// TIA Portal V21 program export: 0 tag tables, 0 data types, 38 data blocks, 68 code blocks (in call order from the OBs), 32 instance data blocks

DATA_BLOCK "HmiTags"   // DB16
{ S7_Optimized_Access := 'FALSE' }
// stored: AutoNumber false
   VAR
      MasterReset : Bool;
      SystemRestart : Bool;
      ManualModeFAULT : Bool;
      AlarmAck : Bool;
      Hooter : Bool;
      ResetButton : Bool;
      VesselStatus : Int;
      Weight_int : Int;
      Weight_Temp : Real;
      VesselMaxPressure : Real := 5.0;
      CycleDataLog : Bool;
      CyclePrintData : Bool;
      AlarmPath : String := '/media/simatic/data-storage/Reports/Pdf/Alarm.pdf';
      HelpPath : String := ' /media/simatic/data-storage/OPM/R-OPM.pdf';
      AlarmStarTime : DTL;
      AlarmEndTime : DTL;
      EpoxyMMActual { S7_SetPoint := 'True'} : Real;
      PlcHmiComBreak : Bool;
      AuditStartTime : DTL;
      AuditEndTime : DTL;
      AuditPath : String := '/media/simatic/data-storage/Reports/Pdf/Audit.pdf';
      UserAuditStartTime : DTL;
      UserAuditEndTime : DTL;
      UserAuditPath : String := '/media/simatic/data-storage/Reports/Pdf/UserAudit.pdf';
      LF_time_delay : Int;
      JacketRecoveryCycSelected : Bool;
      JacketRecoveryFault : Bool;
      JacketRecoveryCycEnable : Bool;
      pulse : Array[0..14] of Bool;
      BatchDetailsBlankPopup : Bool;
      BatchDetailsBlankPopupAck : Bool;
      AccessTablePath : String := '/media/simatic/data-storage/Reports/Pdf/AccessTable.pdf';
      LoadCellResult : String;
   END_VAR
BEGIN
END_DATA_BLOCK

DATA_BLOCK "LifeBeatMonitor"   // DB153
{ S7_Optimized_Access := 'FALSE' }
// stored: AutoNumber false
   VAR
      CommunicationBits : Word;
      LifeBit : Bool;
      OnlineOfflineBeat : Bool;
      StartupBit : Bool;
   END_VAR
BEGIN
END_DATA_BLOCK

DATA_BLOCK "ModeDb"   // DB100
{ S7_Optimized_Access := 'FALSE' }
// stored: AutoNumber false
   VAR
      Cycle1 { S7_SetPoint := 'True'} : "ModePara";   // PHT
      Cycle2 { S7_SetPoint := 'True'} : "ModePara";   // BATCH
      Cycle3 { S7_SetPoint := 'True'} : "ModePara";   // SIP
      Cycle4 { S7_SetPoint := 'True'} : "ModePara";   // CIP
      Cycle5 { S7_SetPoint := 'True'} : "ModePara";   // LOAD CELL CALIBRATION
      VesselWeight { S7_SetPoint := 'True'} : Real;
      AlarmStarTime : DTL;
      AlarmEndTime : DTL;
   END_VAR
BEGIN
   Cycle2.CycleName := 'BATCH';
   Cycle3.CycleName := 'SIP';
   Cycle4.CycleName := 'CIP';
   Cycle5.CycleName := 'BULKSTRL';
END_DATA_BLOCK

DATA_BLOCK "ModeDb_R"   // DB110
{ S7_Optimized_Access := 'FALSE' }
// stored: AutoNumber false
   VAR RETAIN
      ManualMode : "ManualModePara";   // MANUAL MODE
      RunningCycle { S7_SetPoint := 'True'} : "CycleDetails";
      BaseReportPath : String := '/media/simatic/data-storage/Reports/Pdf/';
      FinalReportPath : String;
      ReportId : Int;
      Cycle1 { S7_SetPoint := 'True'} : "ModeParaR";   // PHT
      Cycle2 { S7_SetPoint := 'True'} : "ModeParaR";   // BATCH
      Cycle3 { S7_SetPoint := 'True'} : "ModeParaR";   // SIP
      Cycle4 { S7_SetPoint := 'True'} : "ModeParaR";   // CIP
      Cycle5 { S7_SetPoint := 'True'} : "ModeParaR";   // LOAD CELL CALIBRATION
      ReportName : String[100];
   END_VAR
BEGIN
   RunningCycle.PrintInterval := 30;
END_DATA_BLOCK

DATA_BLOCK "ProcessAlarms"   // DB191
{ S7_Optimized_Access := 'FALSE' }
// stored: AutoNumber false
   VAR
      CipCycleOver : Bool;
      CipCycleConductivityReached : Bool;
      CipCycleConductivityNotReached : Bool;
      ConductivityNotSampled : Bool;
      CipReportDataNotLogged : Bool;
      PhtFailed : Bool;
      PhtPassed : Bool;
      PhtOver : Bool;
      PhtReportDataNotLogged : Bool;
      SterilizationTimeOver : Bool;
      SteamFlowLow : Bool;
      SterilizationHighTemperature : Bool;
      SterilizationCycleCompleted : Bool;
      SterilizationReportDataNotLogged : Bool;
      WfiFlowLow : Bool;
      BatchWfiFlowLow : Bool;
   END_VAR
BEGIN
END_DATA_BLOCK

DATA_BLOCK "SafetyAlarms"   // DB181
{ S7_Optimized_Access := 'FALSE' }
// stored: AutoNumber false
   VAR
      ControlKeyOff : Bool;
      EmergencyStopPressed : Bool;
      PowerReset : Bool;
      CompresseDairPressurelow : Bool;
      PowerFailure : Bool;
      PlcRestarted : Bool;
      Mm01FeedbackTrip : Bool;
      Cp01FeedbackTrip : Bool;
      Mm01OverloadTrip : Bool;
      Cp01OverloadTrip : Bool;
      MinimumWeightRequiredToStartmm01 : Bool;
      Ticr01WireBreak : Bool;
      Ticr02WireBreak : Bool;
      Ticr03WireBreak : Bool;
      Ticr04WireBreak : Bool;
      Ticr05WireBreak : Bool;
      Ticr06WireBreak : Bool;
      Ticr07WireBreak : Bool;
      Ticr08WireBreak : Bool;
      Ticr09WireBreak : Bool;
      Ticr10WireBreak : Bool;
      Picr01WireBreak : Bool;
      Picr02WireBreak : Bool;
      Picr03WireBreak : Bool;
      Picr04WireBreak : Bool;
      Cicr01WireBreak : Bool;
      Lc01CommunicationFailed : Bool;
      VesselHighPressure : Bool;
      Mm01SpeedSensorTrip : Bool;
      PlcToHmiCommunicationFailed : Bool;
   END_VAR
BEGIN
END_DATA_BLOCK

DATA_BLOCK "TimerAlarm"   // DB185
{ S7_Optimized_Access := 'FALSE' }
// stored: AutoNumber false
   VAR
      ControlKeyOff : IEC_TIMER;
      EmergencyStopPressed : IEC_TIMER;
      PowerReset : IEC_TIMER;
      CompresseDairPressurelow : IEC_TIMER;
      PowerFailure : IEC_TIMER;
      PlcRestarted : IEC_TIMER;
      Mm01FeedbackTrip : IEC_TIMER;
      Cp01FeedbackTrip : IEC_TIMER;
      Mm01OverloadTrip : IEC_TIMER;
      Cp01OverloadTrip : IEC_TIMER;
      MinimumWeightRequiredToStartmm01 : IEC_TIMER;
      Ticr01WireBreak : IEC_TIMER;
      Ticr02WireBreak : IEC_TIMER;
      Ticr03WireBreak : IEC_TIMER;
      Ticr04WireBreak : IEC_TIMER;
      Ticr05WireBreak : IEC_TIMER;
      Ticr06WireBreak : IEC_TIMER;
      Ticr07WireBreak : IEC_TIMER;
      Ticr08WireBreak : IEC_TIMER;
      Ticr09WireBreak : IEC_TIMER;
      Ticr10WireBreak : IEC_TIMER;
      Picr01WireBreak : IEC_TIMER;
      Picr02WireBreak : IEC_TIMER;
      Picr03WireBreak : IEC_TIMER;
      Picr04WireBreak : IEC_TIMER;
      Cicr01WireBreak : IEC_TIMER;
      Lc01CommunicationFailed : IEC_TIMER;
      VesselHighPressure : IEC_TIMER;
      Mm01SpeedSensorTrip : IEC_TIMER;
      PlcToHmiCommunicationFailed : IEC_TIMER;
      CipCycleOver : IEC_TIMER;
      CipCycleConductivityReached : IEC_TIMER;
      CipCycleConductivityNotReached : IEC_TIMER;
      ConductivityNotSampled : IEC_TIMER;
      CipReportDataNotLogged : IEC_TIMER;
      PhtFailed : IEC_TIMER;
      PhtPass : IEC_TIMER;
      PhtOver : IEC_TIMER;
      PhtReportDataNotLogged : IEC_TIMER;
      SterilizationTimeOver : IEC_TIMER;
      SteamFlowLow : IEC_TIMER;
      SterilizationHighTemperature : IEC_TIMER;
      SterilizationCycleCompleted : IEC_TIMER;
      SterilizationReportDataNotLogged : IEC_TIMER;
      WfiFlowLow : IEC_TIMER;
      BatchReportDataNotLogged : IEC_TIMER;
      LifeBitAlarm { S7_SetPoint := 'True'} : IEC_TIMER;
      AlarmAck_Reset { S7_SetPoint := 'True'} : IEC_TIMER;
      MasterReset { S7_SetPoint := 'True'} : IEC_TIMER;
   END_VAR
BEGIN
END_DATA_BLOCK

DATA_BLOCK "pulse"   // DB8
{ S7_Optimized_Access := 'FALSE' }
   VAR
      ControlKeyOff : Bool;
      EmergencyStopPressed : Bool;
      PowerReset : Bool;
      CompresseDairPressurelow : Bool;
      PowerFailure : Bool;
      PlcRestarted : Bool;
      Mm01FeedbackTrip : Bool;
      Cp01FeedbackTrip : Bool;
      Mm01OverloadTrip : Bool;
      Cp01OverloadTrip : Bool;
      MinimumWeightRequiredToStartmm01 : Bool;
      Ticr01WireBreak : Bool;
      Ticr02WireBreak : Bool;
      Ticr03WireBreak : Bool;
      Ticr04WireBreak : Bool;
      Ticr05WireBreak : Bool;
      Ticr06WireBreak : Bool;
      Ticr07WireBreak : Bool;
      Ticr08WireBreak : Bool;
      Ticr09WireBreak : Bool;
      Ticr10WireBreak : Bool;
      Picr01WireBreak : Bool;
      Picr02WireBreak : Bool;
      Picr03WireBreak : Bool;
      Picr04WireBreak : Bool;
      Cicr01WireBreak : Bool;
      Lc01CommunicationFailed : Bool;
      VesselHighPressure : Bool;
      Mm01SpeedSensorTrip : Bool;
      PlcToHmiCommunicationFailed : Bool;
      CipCycleOver : Bool;
      CipCycleConductivityReached : Bool;
      CipCycleConductivityNotReached : Bool;
      ConductivityNotSampled : Bool;
      CipReportDataNotLogged : Bool;
      PhtFailed : Bool;
      PhtPass : Bool;
      PhtOver : Bool;
      PhtReportDataNotLogged : Bool;
      SterilizationTimeOver : Bool;
      SteamFlowLow : Bool;
      SterilizationHighTemperature : Bool;
      SterilizationCycleCompleted : Bool;
      SterilizationReportDataNotLogged : Bool;
      WfiFlowLow : Bool;
      BatchReportDataNotLogged : Bool;
   END_VAR
BEGIN
END_DATA_BLOCK

DATA_BLOCK "BatchRe"   // DB33
{ S7_Optimized_Access := 'TRUE' }
// stored: AutoNumber false, MemoryReserve 100
   VAR
      ReBit : Array[0..20] of Bool;
      BatchLinePrint : Array[0..60] of String;
   END_VAR
BEGIN
   BatchLinePrint[1] := 'BATCH STARTED';
   BatchLinePrint[2] := 'BATCH OVER';
   BatchLinePrint[3] := 'FILL WFI STARTED';
   BatchLinePrint[4] := 'FILL WFI PAUSED';
   BatchLinePrint[5] := 'FILL WFI RESUMED';
   BatchLinePrint[6] := 'FILL WFI OVER';
   BatchLinePrint[7] := 'FILL WFI RESET';
   BatchLinePrint[8] := 'TEMPERATURE CONTROL HEATING STARTED';
   BatchLinePrint[9] := 'TEMPERATURE CONTROL COOLING STARTED';
   BatchLinePrint[10] := 'TEMPERATURE CONTROL PAUSED';
   BatchLinePrint[11] := 'TEMPERATURE CONTROL RESUMED';
   BatchLinePrint[12] := 'TEMPERATURE CONTROL HEATING REACHED';
   BatchLinePrint[13] := 'TEMPERATURE CONTROL RESET';
   BatchLinePrint[14] := 'MM01 MIXING STARTED';
   BatchLinePrint[15] := 'MM01 MIXING PAUSED';
   BatchLinePrint[16] := 'MM01 MIXING RESUMED';
   BatchLinePrint[17] := 'MM01 MIXING OVER';
   BatchLinePrint[18] := 'MM01 MIXING RESET';
   BatchLinePrint[19] := 'PRODUCT RECIRCULATION STARTED';
   BatchLinePrint[20] := 'PRODUCT RECIRCULATION PAUSED';
   BatchLinePrint[21] := 'PRODUCT RECIRCULATION RESUMED';
   BatchLinePrint[22] := 'PRODUCT RECIRCULATION OVER';
   BatchLinePrint[23] := 'PRODUCT RECIRCULATION RESET';
   BatchLinePrint[24] := 'MANUAL RM ADDITION STARTED';
   BatchLinePrint[25] := 'MANUAL RM ADDITION PAUSED';
   BatchLinePrint[26] := 'MANUAL RM ADDITION RESUMED';
   BatchLinePrint[27] := 'MANUAL RM ADDITION OVER';
   BatchLinePrint[28] := 'MANUAL RM ADDITION RESET';
   BatchLinePrint[29] := 'N2 SPARGING STARTED';
   BatchLinePrint[30] := 'N2 SPARGING PAUSED';
   BatchLinePrint[31] := 'N2 SPARGING RESUMED';
   BatchLinePrint[32] := 'N2 SPARGING OVER';
   BatchLinePrint[33] := 'N2 SPARGING RESET';
   BatchLinePrint[34] := 'GAS BLANKETING STARTED';
   BatchLinePrint[35] := 'GAS BLANKETING PAUSED';
   BatchLinePrint[36] := 'GAS BLANKETING RESUMED';
   BatchLinePrint[37] := 'GAS BLANKETING RESET';
   BatchLinePrint[38] := 'FINAL VOLUME MAKEUP STARTED';
   BatchLinePrint[39] := 'FINAL VOLUME MAKEUP PAUSED';
   BatchLinePrint[40] := 'FINAL VOLUME MAKEUP RESUMED';
   BatchLinePrint[41] := 'FINAL VOLUME MAKEUP OVER';
   BatchLinePrint[42] := 'FINAL VOLUME MAKEUP RESET';
   BatchLinePrint[43] := 'PRODUCT TRANSFER STARTED';
   BatchLinePrint[44] := 'PRODUCT TRANSFER PAUSED';
   BatchLinePrint[45] := 'PRODUCT TRANSFER RESUMED';
   BatchLinePrint[46] := 'PRODUCT TRANSFER OVER';
   BatchLinePrint[47] := 'PRODUCT TRANSFER RESET';
   BatchLinePrint[48] := 'JACKET VENT OPEN';
   BatchLinePrint[49] := 'JACKET VENT CLOSE';
   BatchLinePrint[50] := 'JACKET DRAIN OPEN';
   BatchLinePrint[51] := 'JACKET DRAIN CLOSE';
   BatchLinePrint[52] := 'TEMPERATURE CONTROL COOLING REACHED';
   BatchLinePrint[53] := '-';
END_DATA_BLOCK

DATA_BLOCK "BatchSAD"   // DB301
{ S7_Optimized_Access := 'FALSE' }
// stored: AutoNumber false
   VAR RETAIN
      BatchStart : Bool;
      BatchEnd : Bool;
      BatchStartPopup : Bool;
      BatchStartPopupYes : Bool;
      BatchStartPopupNo : Bool;
      BatchEndPopup : Bool;
      BatchEndPopupYes : Bool;
      BatchEndPopupNo : Bool;
      Fault : Bool;
      RmAddVesselSafetyPressurePopup : Bool;
      BatchEventString : String;
      BatchStartPopup2 : Bool;
      BatchStartPopup2Ack : Bool;
      ProdTransferFilterSel : Int;   // 0 - FILTER BYPASS 1- THROUGH PF01 2- THROUGH PF02
   END_VAR
BEGIN
END_DATA_BLOCK

DATA_BLOCK "BatchTimer"   // DB315
{ S7_Optimized_Access := 'TRUE' }
// stored: AutoNumber false, MemoryReserve 100
   VAR
      Timer01 : IEC_TIMER;
      Timer02 { S7_SetPoint := 'True'} : IEC_TIMER;
      Timer03 { S7_SetPoint := 'True'} : IEC_TIMER;
      Timer04 { S7_SetPoint := 'True'} : IEC_TIMER;
      Timer05 { S7_SetPoint := 'True'} : IEC_TIMER;
      Timer06 { S7_SetPoint := 'True'} : IEC_TIMER;
      Timer07 { S7_SetPoint := 'True'} : IEC_TIMER;
      Timer08 { S7_SetPoint := 'True'} : IEC_TIMER;
      Timer09 { S7_SetPoint := 'True'} : IEC_TIMER;
      Timer10 { S7_SetPoint := 'True'} : IEC_TIMER;
      Timer11 { S7_SetPoint := 'True'} : IEC_TIMER;
      Timer12 { S7_SetPoint := 'True'} : IEC_TIMER;
      Timer13 { S7_SetPoint := 'True'} : IEC_TIMER;
      Timer14 { S7_SetPoint := 'True'} : IEC_TIMER;
      Timer15 { S7_SetPoint := 'True'} : IEC_TIMER;
      Timer16 { S7_SetPoint := 'True'} : IEC_TIMER;
      Timer17 { S7_SetPoint := 'True'} : IEC_TIMER;
      Timer18 { S7_SetPoint := 'True'} : IEC_TIMER;
      Timer19 { S7_SetPoint := 'True'} : IEC_TIMER;
      Timer20 { S7_SetPoint := 'True'} : IEC_TIMER;
      Timer21 { S7_SetPoint := 'True'} : IEC_TIMER;
      Timer22 { S7_SetPoint := 'True'} : IEC_TIMER;
      Timer23 { S7_SetPoint := 'True'} : IEC_TIMER;
      Timer24 { S7_SetPoint := 'True'} : IEC_TIMER;
      Timer25 { S7_SetPoint := 'True'} : IEC_TIMER;
      Timer26 { S7_SetPoint := 'True'} : IEC_TIMER;
      Timer27 { S7_SetPoint := 'True'} : IEC_TIMER;
      Timer28 { S7_SetPoint := 'True'} : IEC_TIMER;
      Timer29 { S7_SetPoint := 'True'} : IEC_TIMER;
      Timer30 { S7_SetPoint := 'True'} : IEC_TIMER;
      Timer31 { S7_SetPoint := 'True'} : IEC_TIMER;
      Timer32 { S7_SetPoint := 'True'} : IEC_TIMER;
      Timer33 { S7_SetPoint := 'True'} : IEC_TIMER;
      Timer34 { S7_SetPoint := 'True'} : IEC_TIMER;
      Timer35 { S7_SetPoint := 'True'} : IEC_TIMER;
      Timer36 { S7_SetPoint := 'True'} : IEC_TIMER;
      Timer37 { S7_SetPoint := 'True'} : IEC_TIMER;
      Timer38 { S7_SetPoint := 'True'} : IEC_TIMER;
      Timer39 { S7_SetPoint := 'True'} : IEC_TIMER;
      Timer40 { S7_SetPoint := 'True'} : IEC_TIMER;
      Timer41 { S7_SetPoint := 'True'} : IEC_TIMER;
      Timer42 { S7_SetPoint := 'True'} : IEC_TIMER;
      Timer43 { S7_SetPoint := 'True'} : IEC_TIMER;
      Timer44 { S7_SetPoint := 'True'} : IEC_TIMER;
      Timer45 { S7_SetPoint := 'True'} : IEC_TIMER;
      Timer46 { S7_SetPoint := 'True'} : IEC_TIMER;
      Timer47 { S7_SetPoint := 'True'} : IEC_TIMER;
      Timer48 { S7_SetPoint := 'True'} : IEC_TIMER;
      Timer49 { S7_SetPoint := 'True'} : IEC_TIMER;
      Timer50 { S7_SetPoint := 'True'} : IEC_TIMER;
      Timer51 { S7_SetPoint := 'True'} : IEC_TIMER;
      Timer52 { S7_SetPoint := 'True'} : IEC_TIMER;
      Timer53 { S7_SetPoint := 'True'} : IEC_TIMER;
      Timer54 { S7_SetPoint := 'True'} : IEC_TIMER;
      Timer55 { S7_SetPoint := 'True'} : IEC_TIMER;
      Timer56 { S7_SetPoint := 'True'} : IEC_TIMER;
      Timer57 { S7_SetPoint := 'True'} : IEC_TIMER;
      Timer58 { S7_SetPoint := 'True'} : IEC_TIMER;
      Timer59 { S7_SetPoint := 'True'} : IEC_TIMER;
      Timer60 { S7_SetPoint := 'True'} : IEC_TIMER;
      Timer61 { S7_SetPoint := 'True'} : IEC_TIMER;
      Timer62 { S7_SetPoint := 'True'} : IEC_TIMER;
      Timer63 { S7_SetPoint := 'True'} : IEC_TIMER;
      Timer64 { S7_SetPoint := 'True'} : IEC_TIMER;
      Timer65 { S7_SetPoint := 'True'} : IEC_TIMER;
   END_VAR
BEGIN
END_DATA_BLOCK

DATA_BLOCK "CipDo"   // DB202
{ S7_Optimized_Access := 'FALSE' }
// stored: AutoNumber false
   VAR
      MM01CmdMagneticMixerMvCommand : Bool;
      CP01CmdCentrifugalPumpMvAreaCommand : Bool;
      HTR01HooterMvArea : Bool;
      LF01VesselLampOutputMv1000 : Bool;
      SPARE4 : Bool;
      SPARE5 : Bool;
      SPARE6 : Bool;
      SPARE7 : Bool;
   END_VAR
BEGIN
END_DATA_BLOCK

DATA_BLOCK "CipPulse"   // DB204
{ S7_Optimized_Access := 'FALSE' }
// stored: AutoNumber false
   VAR
      RE : Array[0..25] of Bool;
      D500EventsTimer : Array[0..25] of IEC_TIMER;
   END_VAR
BEGIN
END_DATA_BLOCK

DATA_BLOCK "CipTimer"   // DB637
{ S7_Optimized_Access := 'TRUE' }
// stored: AutoNumber false, MemoryReserve 100
   VAR
      Timer1 : IEC_TIMER;
      Timer2 { S7_SetPoint := 'True'} : IEC_TIMER;
      Timer3 { S7_SetPoint := 'True'} : IEC_TIMER;
      Timer4 { S7_SetPoint := 'True'} : IEC_TIMER;
      Timer5 { S7_SetPoint := 'True'} : IEC_TIMER;
   END_VAR
BEGIN
END_DATA_BLOCK

DATA_BLOCK "DateTime"   // DB118
{ S7_Optimized_Access := 'FALSE' }
// stored: AutoNumber false
   VAR
      time_local_read : DTL;
      time_system_read : DTL;
      time_system_write : DTL;
      local_time : Int := 0;
      read_system_time : Int;
      write_system_time : Int;
      write_time : Bool := false;
      write_time_re : Bool;
      time_local_read_ReportName : DTL;
   END_VAR
BEGIN
END_DATA_BLOCK

DATA_BLOCK "RTC_to_String_Conversion Block"   // DB119
{ S7_Optimized_Access := 'TRUE' }
// stored: AutoNumber false, MemoryReserve 100
   VAR
      date_int : Int;
      date_string : String[6];
      month_int : Int;
      month_string : String[6];
      year_string : String[6];
      hour_int : Int;
      hour_string : String[6];
      minute_int : Int;
      minute_string : String[6];
      second_int : Int;
      second_string : String[6];
      date_temp : String[6];
      date_zero : Int;
      date_actual : String[12];
      month_temp : String[6];
      month_zero : Int;
      month_actual : String[6];
      year_actual : String[6];
      hour_temp : String[6];
      hour_zero : Int;
      hour_actual : String[6];
      minute_temp : String[6];
      minute_zero : Int;
      minute_actual : String[6];
      second_temp : String[6];
      second_zero : Int;
      second_actual : String[12];
      Final_Date : String[12];
      Final_time_HRS : String[12];
      Final_time_MINS : String[12];
      Final_time_1 : String[12];
      Final_time : String[8];
      SPACE : String[10];
   END_VAR
BEGIN
END_DATA_BLOCK

DATA_BLOCK "Ai_Faceplate_Db"   // DB107
{ S7_Optimized_Access := 'TRUE' }
// stored: AutoNumber false, MemoryReserve 100
   VAR
      Ai01 : "Ai_Faceplate";   // Ticr01NfcoLineTemp
      Ai02 : "Ai_Faceplate";   // Ticr02VfcoLineTemp
      Ai03 : "Ai_Faceplate";   // Ticr03SvcoLineTemp
      Ai04 : "Ai_Faceplate";   // Ticr04VdcoTemp
      Ai05 : "Ai_Faceplate";   // Ticr05CipPumpDrainTemp
      Ai06 : "Ai_Faceplate";   // Ticr06Pf01InLineTemp
      Ai07 : "Ai_Faceplate";   // Ticr07Pf02InLineTemp
      Ai08 : "Ai_Faceplate";   // Ticr08Pf02OutLineTemp
      Ai09 : "Ai_Faceplate";   // Ticr09PtlDrainTemp
      Ai10 : "Ai_Faceplate";   // Ticr10VesselTemp
      Ai11 : "Ai_Faceplate";   // Picr01VesselPressure
      Ai12 : "Ai_Faceplate";   // Picr02VesselRclLine
      Ai13 : "Ai_Faceplate";   // Picr03Pf01OutLinePressure
      Ai14 : "Ai_Faceplate";   // Picr04Pf02OutLinePressure
      Ai15 : "Ai_Faceplate";   // Cicr01ProcessDrainConductivity
      Ai16 : "Ai_Faceplate";   // AiSpare1
      Ai17 : "Ai_Faceplate";   // AiSpare2
      Ai18 : "Ai_Faceplate";   // AiSpare3
      Ai19 : "Ai_Faceplate";   // AiSpare4
      Ai20 : "Ai_Faceplate";   // AiSpare5
      Ai21 : "Ai_Faceplate";   // AiSpare6
      Ai22 : "Ai_Faceplate";   // AiSpare7
      Ai23 : "Ai_Faceplate";   // AiSpare8
      Ai24 : "Ai_Faceplate";   // AiSpare9
      Ai25 : "Ai_Faceplate";
      Ai26 : "Ai_Faceplate";
   END_VAR
BEGIN
END_DATA_BLOCK

DATA_BLOCK "Ao_Faceplate_Db"   // DB105
{ S7_Optimized_Access := 'FALSE' }
// stored: AutoNumber false
   VAR
      Mm01Ref : "Ao_Faceplate";
      Cp01Ref : "Ao_Faceplate";
      Cv01 : "Ao_Faceplate";
      AoSpare1 : "Ao_Faceplate";
      AoSpare2 : "Ao_Faceplate";
      AoSpare3 : "Ao_Faceplate";
      AoSpare4 : "Ao_Faceplate";
      AoSpare5 : "Ao_Faceplate";
   END_VAR
BEGIN
END_DATA_BLOCK

DATA_BLOCK "DO_FaceplateDb"   // DB101
{ S7_Optimized_Access := 'FALSE' }
// stored: AutoNumber false
   VAR
      Cv01 : "Do_Faceplate";
      Cv02 : "Do_Faceplate";
      Cv03 : "Do_Faceplate";
      Cv04 : "Do_Faceplate";
      Cv05 : "Do_Faceplate";
      Cv06 : "Do_Faceplate";
      Cv07 : "Do_Faceplate";
      Cv08 : "Do_Faceplate";
      Cv09 : "Do_Faceplate";
      Cv10 : "Do_Faceplate";
      Cv11 : "Do_Faceplate";
      Cv12 : "Do_Faceplate";
      Cv13 : "Do_Faceplate";
      Cv14 : "Do_Faceplate";
      Cv15 : "Do_Faceplate";
      Cv16 : "Do_Faceplate";
      Cv17 : "Do_Faceplate";
      Cv18 : "Do_Faceplate";
      Cv19 : "Do_Faceplate";
      Cv20 : "Do_Faceplate";
      Cv21 : "Do_Faceplate";
      Cv22 : "Do_Faceplate";
      Cv23 : "Do_Faceplate";
      Cv24 : "Do_Faceplate";
      Cv25 : "Do_Faceplate";
      Cv26 : "Do_Faceplate";
      Cv27 : "Do_Faceplate";
      Cv28 : "Do_Faceplate";
      Cv29 : "Do_Faceplate";
      Cv30 : "Do_Faceplate";
      Cv31 : "Do_Faceplate";
      Cv32 : "Do_Faceplate";
      Cv33 : "Do_Faceplate";
      Cv34 : "Do_Faceplate";
      Cv35 : "Do_Faceplate";
      Cv36 : "Do_Faceplate";
      Cv37 : "Do_Faceplate";
      Cv38 : "Do_Faceplate";
      Cv39 : "Do_Faceplate";
      Cv40 : "Do_Faceplate";
      Cv41 : "Do_Faceplate";
      Cv42 : "Do_Faceplate";
      Cv43 : "Do_Faceplate";
      Cv44 : "Do_Faceplate";
      Cv45 : "Do_Faceplate";
      Cv46 : "Do_Faceplate";
      Cv47 : "Do_Faceplate";
      Cv48 : "Do_Faceplate";
      Cv49 : "Do_Faceplate";
      Cv50 : "Do_Faceplate";
      Cv51 : "Do_Faceplate";
      Cv52 : "Do_Faceplate";
      Cv53 : "Do_Faceplate";
      Cv54 : "Do_Faceplate";
      Cv55 : "Do_Faceplate";
      Cv56 : "Do_Faceplate";
      Cv57 : "Do_Faceplate";
      Cv58 : "Do_Faceplate";
      Cv59 : "Do_Faceplate";
      Cv60 : "Do_Faceplate";
      Cv61 : "Do_Faceplate";
      Cv62 : "Do_Faceplate";
      Cv63 : "Do_Faceplate";
      Cv64 : "Do_Faceplate";
      Fbov01 : "Do_Faceplate";
      "Mm01 Ref" { S7_SetPoint := 'True'} : "Do_Faceplate";
      "Cp01 Ref" { S7_SetPoint := 'True'} : "Do_Faceplate";
   END_VAR
BEGIN
END_DATA_BLOCK

DATA_BLOCK "CV15"   // DB209
{ S7_Optimized_Access := 'TRUE' }
// stored: AutoNumber false, MemoryReserve 100
   VAR
      Tag_IB89 : Byte;
      Tag_IB90 : Byte;
      Tag_IB93 : Byte;
      Tag_IB94 : Byte;
      Tag_IB96 : Byte;
      Tag_IB97 : Byte;
      Tag_IB98 : Byte;
      Tag_MD124 : DInt;
      Tag_MD300 : DInt;
      Tag_MD304 : DInt;
      Tag_MD308 : DInt;
      Tag_MD312 : Real;
      Tag_MD316 : Real;
      Tag_MD320 : DInt;
      Tag_MD324 : DInt;
      Tag_MD340 : DInt;
      Tag_MD344 : DInt;
      Tag_MD348 { ExternalWritable := 'False'} : DInt;
      Tag_MD352 : Real;
      Tag_MD356 : Real;
   END_VAR
BEGIN
END_DATA_BLOCK

DATA_BLOCK "PHT Cycle"   // DB1201
{ S7_Optimized_Access := 'FALSE' }
// stored: AutoNumber false
   VAR
      Start : Bool;
      Stop : Bool;
      Abort : Bool;
      fault : Bool;
      Running : Bool;
      Selected : Bool;
      Actual_Min_Pressure : Real;
      Actual_Max_Pressure : Real;
      "Actual Stabilization Time" : DInt;
      "Actual Pressurise Hold Mins" : DInt;
      "Actual Pressurise Hold Secs" : DInt;
      "PHT Step Status int" : Int;
      "Step Status" : String[50];
      "Event Status" : String[50];
      print_event : Bool;
      "Startup Popup" : Bool;
      "Startup Popup Ack" : Bool;
      "Startup Popup Acked" : Bool;
      "Startup parameter popup" : Bool;
      "Abort Confirmation Popup" : Bool;
      "PHT Result" : Int;
      VesselSel : Int := 1;   // 1=Mv1, 2=Mv2, 3=Mv1&Mv2
      Result : String[50];
      Continue_Button : Bool;
      Abort_Button : Bool;
      "Actual Delay to Open Cai" : Int;
      PhtTemp : Bool;
      HOLD_FAIL : Bool;
      "Startup parameter popup No" : Bool;
      "Startup parameter popup Yes" : Bool;
      "Actual Delay to Open N2I" : Int;
      "N2IControl Valve" : Bool;
      EndOverPopup : Bool;
      EndOverPopupAck : Bool;
      CycleAbortEvent : Bool;
      "Abort confirmation popup Yes" : Bool;
      "Abort confirmation popup No" : Bool;
      InitialPressure : Real;
      FinalPressure : Real;
      HoldStartTimeLog : DTL;
      HoldEndTimeLog : DTL;
      TempTime : Time;
      RoundedTime : Time;
      TempMs : DInt;
      RoundedTime_Pos : Time;
      Hours : Int;
      Minutes : Int;
      Seconds : Int;
      TotalSecondsTag : DInt;
      PhtTimeDifference : Time;
   END_VAR
BEGIN
END_DATA_BLOCK

DATA_BLOCK "PHTRe"   // DB41
{ S7_Optimized_Access := 'TRUE' }
// stored: AutoNumber false, MemoryReserve 100
   VAR
      PhtLinePrintText : Array[0..10] of String[40];
      PhtLinePrint1 : String[40];
      RE : Array[0..20] of Bool;
   END_VAR
BEGIN
   PhtLinePrintText[1] := 'PRESSURIZE STARTED';
   PhtLinePrintText[2] := 'STABILIZE STARTED';
   PhtLinePrintText[3] := 'PRESSURE HOLD STARTED';
   PhtLinePrintText[4] := 'PRESSURE RELEASE STARTED';
   PhtLinePrintText[5] := 'CYCLE PAUSED';
   PhtLinePrintText[6] := 'PHT OVER';
END_DATA_BLOCK

DATA_BLOCK "PhtRecipe"   // DB1218
{ S7_Optimized_Access := 'FALSE' }
// stored: AutoNumber false
   VAR
      HoldPressure : Real := 1.33;
      PressureStabilizeTime : Int := 30;
      AcceptableLeakage : Real := 0.2;
      PressureHoldTime : Int := 1;
      ReleasePressure : Real := 0.1;
   END_VAR
BEGIN
END_DATA_BLOCK

DATA_BLOCK "PhtTimer"   // DB1216
{ S7_Optimized_Access := 'FALSE' }
// stored: AutoNumber false
   VAR
      "ReportData ResetTImer" : IEC_TIMER;
      "TIMER" { S7_SetPoint := 'True'} : IEC_TIMER;
      HVEventsTimer : Array[0..20] of IEC_TIMER;
      PhtTime1 { S7_SetPoint := 'True'} : IEC_TIMER;
      PhtTime2 { S7_SetPoint := 'True'} : IEC_TIMER;
      PhtTime3 { S7_SetPoint := 'True'} : IEC_TIMER;
      PhtTime4 { S7_SetPoint := 'True'} : IEC_TIMER;
      PhtTime5 { S7_SetPoint := 'True'} : IEC_TIMER;
      PhtTime6 { S7_SetPoint := 'True'} : IEC_TIMER;
      PhtTime7 { S7_SetPoint := 'True'} : IEC_TIMER;
      PhtTime8 { S7_SetPoint := 'True'} : IEC_TIMER;
      PhtTime9 { S7_SetPoint := 'True'} : IEC_TIMER;
      PhtTime10 { S7_SetPoint := 'True'} : IEC_TIMER;
   END_VAR
BEGIN
END_DATA_BLOCK

DATA_BLOCK "PidParameters"   // DB58
{ S7_Optimized_Access := 'FALSE' }
   VAR RETAIN
      Fv1_Cv01 : Struct
         "Set Value" : Real;
         P : Real := 8.0;
         I : Real := 80.0;
         D : Real := 0.0;
         Mode : Int;
         Output : Real;
         OutputCoil : Bool;
         State : Int;
         Error : Word;
         Reset : Bool;
         InputValue : Real;
      END_STRUCT;
   END_VAR
BEGIN
END_DATA_BLOCK

DATA_BLOCK "CipRe"   // DB42
{ S7_Optimized_Access := 'TRUE' }
// stored: MemoryReserve 100
   VAR
      CipLinePrintText : Array[0..20] of String;
   END_VAR
BEGIN
   CipLinePrintText[1] := 'PRE RINSE CYCLE - RINSING ON STARTED';
   CipLinePrintText[2] := 'PRE RINSE CYCLE - DRAIN ON STARTED';
   CipLinePrintText[3] := 'PRE RINSE CYCLE - SYSTEM DRAIN STARTED';
   CipLinePrintText[4] := 'PRE RINSE CYCLE - AIR PURGING STARTED';
   CipLinePrintText[5] := 'FILLING CYCLE - FILLING ON STARTED';
   CipLinePrintText[6] := 'FILLING CYCLE - MIXING ON STARTED';
   CipLinePrintText[7] := 'FILLING CYCLE - DRAIN ON STARTED';
   CipLinePrintText[8] := 'FILLING CYCLE - SYSTEM DRAIN STARTED';
   CipLinePrintText[9] := 'FILLING CYCLE - AIR PURGING ON STARTED';
   CipLinePrintText[10] := 'WAITING FOR ACKNOWLEDGE';
   CipLinePrintText[11] := 'CYCLE PAUSED';
   CipLinePrintText[12] := 'CIP CYCLE OVER';
   CipLinePrintText[13] := 'CYCLE RESETED';
   CipLinePrintText[14] := 'FILLING CYCLE - RECIRCULATION STARTED';
   CipLinePrintText[15] := 'FINAL RINSE CYCLE - FILLING ON STARTED';
   CipLinePrintText[16] := 'FINAL RINSE CYCLE - MIXING ON STARTED';
   CipLinePrintText[17] := 'FINAL RINSE CYCLE - DRAIN ON STARTED';
   CipLinePrintText[18] := 'FINAL RINSE CYCLE - SYSTEM DRAIN STARTED';
   CipLinePrintText[19] := 'FINAL RINSE CYCLE - AIR PURGING ON STARTED';
   CipLinePrintText[20] := 'FINAL RINSE CYCLE - RECIRCULATION STARTED';
END_DATA_BLOCK

DATA_BLOCK "DB615"   // DB615
TITLE = DB615
{ S7_Optimized_Access := 'FALSE' }
// CIP GENERAL DB
// stored: AutoNumber false
   VAR RETAIN
      Fault : Bool;
      Running : Bool;
      Selected : Bool;
      NoCycleSelectedInterlock : Bool;
      SelectStep : Bool;
      DelayToTriggerStep : Bool;
      ResetLogic : Bool;
      ProcessOver : Bool;
      TempStep : Int;
      CurrentStep : Int;
      CycleStatus : String[60];
      StepStatus : String[60];
      StepStatusInt : Int;
      Re : Array[0..50] of Bool;
      CycleStarted { S7_SetPoint := 'True'} : "CipCycleStarted";
      CycleOver { S7_SetPoint := 'True'} : "CipCycleOver";
      CycleRunningMV : Bool;
      ApActPressure : Real;
      CheckWeightWfi : Real;
      ScanTimeForFillingWfiTemp : Int;
   END_VAR
BEGIN
END_DATA_BLOCK

DATA_BLOCK "DB621"   // DB621
TITLE = DB619
{ S7_Optimized_Access := 'TRUE' }
// CIP BUTTONS DB
// stored: AutoNumber false, MemoryReserve 0
   VAR
      Start : Bool;
   END_VAR
   VAR RETAIN
      MainPopup1Ack : Bool;
      MainPopup2Ack : Bool;
   END_VAR
BEGIN
END_DATA_BLOCK

DATA_BLOCK "DB622"   // DB622
TITLE = DB620
{ S7_Optimized_Access := 'FALSE' }
// CIP POPUPS
// stored: AutoNumber false
   VAR RETAIN
      NoCycleSelectedPopup : Bool;
      MainPopupMsg1 : Bool;
      MainPopupMsg2 : Bool;
   END_VAR
BEGIN
END_DATA_BLOCK

DATA_BLOCK "DB625"   // DB625
TITLE = REPORT PROCESS VALUE
{ S7_Optimized_Access := 'FALSE' }
// stored: AutoNumber false
   VAR RETAIN
      RepetitionPrint : Array[0..3] of Int;
      FillingPrint : Array[0..3] of "FillingPrint";
      MixingTime { S7_SetPoint := 'True'} : Array[0..3] of "MixingPrint";
      Pulsingtime { S7_SetPoint := 'True'} : Array[0..3] of "PulsingPrint";
      spare { S7_SetPoint := 'True'} : Bool;
      RecirculationPrint { S7_SetPoint := 'True'} : Array[0..3] of "RecirculationPrint";
      DrainPrint { S7_SetPoint := 'True'} : Array[0..3] of "DrainPrint";
      ConductivityStatus { S7_SetPoint := 'True'} : Array[0..3] of Bool;
   END_VAR
BEGIN
END_DATA_BLOCK

DATA_BLOCK "DB626"   // DB626
TITLE = ZERO REPORT PROCESS VALUE
{ S7_Optimized_Access := 'FALSE' }
// stored: AutoNumber false
   VAR
      RepetitionPrint : Array[0..3] of Int;
      FillingPrint : Array[0..3] of "FillingPrint";
      MixingTime { S7_SetPoint := 'True'} : Array[0..3] of "MixingPrint";
      Pulsingtime { S7_SetPoint := 'True'} : Array[0..3] of "PulsingPrint";
      spare { S7_SetPoint := 'True'} : Bool;
      RecirculationPrint { S7_SetPoint := 'True'} : Array[0..3] of "RecirculationPrint";
      DrainPrint { S7_SetPoint := 'True'} : Array[0..3] of "DrainPrint";
      ConductivityStatus { S7_SetPoint := 'True'} : Array[0..3] of Bool;
   END_VAR
BEGIN
END_DATA_BLOCK

DATA_BLOCK "DB627"   // DB627
TITLE = SCREEN PROCESS VALUE
{ S7_Optimized_Access := 'FALSE' }
// stored: AutoNumber false
   VAR
      RinseTimeSv : Int;
      RinseTimePv : DInt;
      FillTimeSv : DInt;
      FillTimePv : DInt;
      RepSv : Int;
      RepPv : Int;
      FillQtySv : Real;
      FillQtyPv : Real;
      MixingSv : Int;
      MixingPv : DInt;
      SdSv : Int;
      SdPv : DInt;
      APSv : Int;
      ApPv : DInt;
      ApReleaseTimeSv : Int;
      ApReleaseTimePv : DInt;
      CurrentStepNo : Int;
      CycleStatus : String[60];
      StepStatus : String[60];
      ApSetPressureSv : Real;
      ApSetPressurePv : Real;
      CombineAPSv : Int;
      CombineApPv : DInt;
      CombineApReleaseTimeSv : Int;
      CombineApReleaseTimePv : DInt;
      DosingTimePv : DInt;
      PulsingTimeSv : Int;
      RecirculationSv : Int;
      RecirculationPv : DInt;
      ConductivitySv : Real;
      ConductivityPv : Real;
   END_VAR
BEGIN
END_DATA_BLOCK

DATA_BLOCK "DB616"   // DB616
TITLE = DB616
{ S7_Optimized_Access := 'FALSE' }
// CIP Recipe
// stored: AutoNumber false
   VAR
      TotalStep : Int := 3;
      CycleSelection { S7_SetPoint := 'True'} : Array[0..3] of "CIP";
      MainPopup1Enable : Bool := 1;
      MainPopup2Enable : Bool := 1;
      FillingInputPara { S7_SetPoint := 'True'} : Array[0..3] of "FillingInputs";
      FillingOutputPara { S7_SetPoint := 'True'} : Array[0..3] of "FillingOutputs";
      MixingTimeInput : Array[0..3] of Int;
      RecirculationInput { S7_SetPoint := 'True'} : Array[0..3] of "RecirculationInputs";
      RecirculationOutput { S7_SetPoint := 'True'} : Array[0..3] of "RecirculationOutputs";
      DrainInputs { S7_SetPoint := 'True'} : Array[0..3] of "DrainInputs";
      DrainOutputs : Array[0..3] of "DrainOutputs";
      SystemDrainSetTimeInput : Array[0..3] of Int;
      SystemDrainOutPara { S7_SetPoint := 'True'} : Array[0..3] of "SystemDrainOutputs";
      AirPurgingInputPara { S7_SetPoint := 'True'} : Array[0..3] of "AirPurgingInputs";
      AirPurgingOutPara { S7_SetPoint := 'True'} : Array[0..3] of "AirPurgingOutputs";
      CycleNames : Array[0..3] of String[60];
      Spare : Bool;
   END_VAR
BEGIN
   CycleSelection[0..3].StepSelection.SuctionLineCleanNoYes := 0;
   CycleSelection[0..3].StepSelection.VacuumDryingNoYes := 0;
   CycleSelection[0].StepSelection.FillingNoYes := 0;
   CycleSelection[1..3].StepSelection.FillingNoYes := 1;
   CycleSelection[0..3].StepSelection.TemperatureDosingNoYes := 0;
   CycleSelection[0..3].StepSelection.TransferNoYes := 0;
   CycleSelection[0..1].StepSelection.MIxingNoYes := 0;
   CycleSelection[2..3].StepSelection.MIxingNoYes := 1;
   CycleSelection[0..1].StepSelection.RecirculationNoYes := 0;
   CycleSelection[2..3].StepSelection.RecirculationNoYes := 1;
   CycleSelection[0].StepSelection.DrainNoYes := 0;
   CycleSelection[1..3].StepSelection.DrainNoYes := 1;
   CycleSelection[0].StepSelection.SystemDrainNoYes := 0;
   CycleSelection[1..3].StepSelection.SystemDrainNoYes := 1;
   CycleSelection[0].StepSelection.AirPurgingNoYes := 0;
   CycleSelection[1..3].StepSelection.AirPurgingNoYes := 1;
   CycleSelection[1..3].StepSelection.ConductivityCheckWhileRinse := 0;
   CycleSelection[0..2].StepSelection.ConductivityCheckWhileDrain := 0;
   CycleSelection[3].StepSelection.ConductivityCheckWhileDrain := 1;
   CycleSelection[0..2].StepSelection.SetRepetition := 0;
   CycleSelection[0..3].StepSelection.TimeSaveModeNoYes := 0;
   CycleSelection[1].StepSelection.ConductivityCheckWhileTransfer := false;
   CycleSelection[2..3].StepSelection.ConductivityCheckWhileTransfer := 0;
   FillingInputPara[1].Selections.FillMethodSel := 3;
   FillingInputPara[2..3].Selections.FillMethodSel := 0;
   FillingInputPara[1..3].Selections.FillTimeBaseSel := 0;
   FillingInputPara[0].Selections.UtilitySel := 1;
   FillingInputPara[1..3].Selections.UtilitySel := 2;
   FillingInputPara[1..3].Selections.ConductivityWhileRinse := 0;
   FillingInputPara[0].Selections.RinseCondition := 1;
   FillingInputPara[1..3].Selections.RinseCondition := 0;
   FillingInputPara[1].Selections.BypassRinseCondition := 1;
   FillingInputPara[2..3].Selections.BypassRinseCondition := 0;
   FillingInputPara[1..3].Selections.BypassWeightWhileRinseCycle := 0;
   FillingInputPara[0..3].Selections.SeperateParaForRep := 1;
   FillingInputPara[1..2].ProductionSetting.LoopDelay1 := 0;
   FillingInputPara[1].ProductionSetting.ZDVDelay := 0;
   FillingInputPara[0].PreciseEngineering.Loops := 1;
   FillingInputPara[1].PreciseEngineering.Loops := 16;
   FillingInputPara[2..3].PreciseEngineering.Loops := 5;
   FillingInputPara[1..3].PreciseEngineering.VesselMaxWeight := 3000.0;
   MixingTimeInput[2..3] := 1;
   RecirculationInput[2..3].Selections.PressureModeSel := 0;
   RecirculationInput[2..3].Selections.PumpSel := 0;
   RecirculationInput[2].Parameters.RecirculationInputToRunTime := 0;
   RecirculationInput[1].PreciseEngineering.Loops := 0;
   RecirculationInput[2..3].PreciseEngineering.Loops := 5;
   DrainInputs[0..3].Selections.DrainMethodSel := 0;
   DrainInputs[1..3].Selections.PressureModeSel := 1;
   DrainInputs[1].Selections.DrainPumpSel := 0;
   DrainInputs[2..3].Selections.DrainPumpSel := 1;
   DrainInputs[0..1].Selections.InputToRunPump := 0;
   DrainInputs[2..3].Selections.InputToRunPump := 1;
   DrainInputs[1..2].Selections.ConductivityWhileDrain := 0;
   DrainInputs[3].Selections.ConductivityWhileDrain := 1;
   DrainInputs[1..2].Selections.ConductivityWhileDrainPTL := 0;
   DrainInputs[1..2].Selections.CipSkidWeightSel := 0;
   DrainInputs[1..2].Selections.MultiConductivityCheck := 0;
   DrainInputs[0..1].PreciseEngineering.Loops := 1;
   DrainInputs[2..3].PreciseEngineering.Loops := 10;
   AirPurgingInputPara[1..3].Selections.ApMethod := 0;
   AirPurgingInputPara[1..3].Selections.PressureMode := 1;
   AirPurgingInputPara[1..3].Selections.VentBeforeOver := 1;
   AirPurgingInputPara[1..3].Selections.AirPurgingSel := 0;
   AirPurgingInputPara[1..3].PreciseEngineering.Loops := 17;
   CycleNames[1] := 'PRE RINSE CYCLE';
   CycleNames[2] := 'FILLING CYCLE';
   CycleNames[3] := 'FINAL RINSE CYCLE';
END_DATA_BLOCK

DATA_BLOCK "DB623"   // DB623
TITLE = DB618
{ S7_Optimized_Access := 'FALSE' }
// Recipe
// stored: AutoNumber false
   VAR RETAIN
      StepEnable : Array[0..5] of Bool;
      Mm01Speed : Real := 1200.0;
      Cp01Speed : Real := 1000.0;
      DrainPressure : Real := 1.11;
      AirPurgingPressure : Real := 1.33;
      SystemDrainTime : Int := 30;
      PreRinseCycleSelection : Int := 1;
      FillingCycleSelection : Int := 1;
      FinalRinseCycleSelection : Int := 1;
      PreRinseCycleNoOfRep : Int := 1;
      FillingCycleNoOfRep : Int := 2;
      FillingCycleMixingTime : Int := 30;
      FinalRinseCycleMixingTime : Int := 35;
      FillingCycleFillQty : Real := 500.0;
      FinalRinseCycleFillQty : Real := 1000.0;
      PreRinseCycleSelString : String[10];
      FillingCycleSelString : String[10];
      FinalRinseCycleSelString : String[10];
      FinalRinseSetCond : Real := 1.22;
      SbiOnTime : Int := 10;
      SbiOffTime : Int := 5;
   END_VAR
BEGIN
   StepEnable[0] := FALSE;
   StepEnable[1..3] := TRUE;
END_DATA_BLOCK

DATA_BLOCK "DB624"   // DB624
{ S7_Optimized_Access := 'FALSE' }
// stored: AutoNumber false
   VAR RETAIN
      PcdTime : Int := 10;
      VesselDrainWeight : Real := 15.0;
      AirPurgingPressureTolerence : Real := 0.1;
      AirPurgingReleaseTime : Int := 30;
      DrainPressureTolerance : Real := 0.2;
      DelayToCheckConductivity : Int := 10;
      ConductivityCheckTime : Int := 5;
      "FinalRinseCycleNo.OfRep" : Int := 3;
      FillRinseSamplingLineDelay : Int := 30;
      FillRinseBlanketingLineDelay : Int := 30;
      FillRinseJTubeLineDelay : Int := 30;
      FillRinseSpargingLineDelay : Int := 30;
      FillRinseSbiLineDelay : Int := 30;
      FillRinseRecirculationlineDelay : Int := 30;
      FillRinseVesselBypassLineDelay : Int := 30;
      FillRinsePumpBypassLineDelay : Int := 30;
      FillRinsePf01InLineDelay : Int := 30;
      FillRinsePf01VentLineDelay : Int := 30;
      FillRinsePf02InLineDelay : Int := 30;
      FillRinsePf02VentLineDelay : Int := 30;
      FillRinsePf02OutLineDelay : Int := 30;
      FillRinsePf01BypassLineDelay : Int := 30;
      FillRinsePf02BypassLineDelay : Int := 30;
      FillRinsePtlLineDelay : Int := 30;
      RecSamplingLineDelay : Int := 30;
      RecBlanketingLineDelay : Int := 30;
      RecJTubeLineDelay : Int := 30;
      RecSpargingLineDelay : Int := 30;
      RecSbiLineDelay : Int := 30;
      DrainVesselDrainLineDelay : Int := 30;
      DrainPumpBypassLineDelay : Int := 30;
      DrainPf01InLineDelay : Int := 30;
      DrainPf01VentLineDelay : Int := 30;
      DrainPf02InLineDelay : Int := 30;
      DrainPf02VentLineDelay : Int := 30;
      DrainPf02OutLineDelay : Int := 30;
      DrainPf01BypassLineDelay : Int := 30;
      DrainPf02BypassLineDelay : Int := 30;
      FinalRinseCycleVesselDrainLineDelay : Int := 30;
      AirPurgeSamplingLineDelay : Int := 30;
      AirPurgeBlankeingLineDelay : Int := 30;
      AirPurgeJTubeLineDelay : Int := 30;
      AirPurgeSpargingLineDelay : Int := 30;
      AirPurgeSbiLineDelay : Int := 30;
      AirPurgeRecirculationlineDelay : Int := 30;
      AirPurgeVesselBypassLineDelay : Int := 30;
      AirPurgeVesselDrainLineDelay : Int := 30;
      AirPurgePumpBypassLineDelay : Int := 30;
      AirPurgePf01InLineDelay : Int := 30;
      AirPurgePf01VentLineDelay : Int := 30;
      AirPurgePf02InLineDelay : Int := 30;
      AirPurgePf02VentLineDelay : Int := 30;
      AirPurgePf02OutLineDelay : Int := 30;
      AirPurgePf01BypassLineDelay : Int := 30;
      AirPurgePf02BypassLineDelay : Int := 30;
      AirPurgePtlLineDelay : Int := 30;
   END_VAR
BEGIN
END_DATA_BLOCK

DATA_BLOCK "DiFinal"   // DB102
{ S7_Optimized_Access := 'FALSE' }
// stored: AutoNumber false
   VAR
      ControlKey : Bool;
      EmergencyStop : Bool;
      CompressedAirPressureLow : Bool;
      PowerFailure : Bool;
      PowerReset : Bool;
      MagneticMixerFeedback : Bool;
      CipPumpFeedback : Bool;
      MagneticMixerOverload : Bool;
      CipPumpOverload : Bool;
      RuptureDisc : Bool;
      Cp01FlowSwitch : Bool;
      DiSpare1 : Bool;
      DiSpare2 : Bool;
      MMHighSpeedSensor : Bool;
      DiSpare3 : Bool;
      DiSpare4 : Bool;
      DiSpare5 : Bool;
      DiSpare6 : Bool;
      DiSpare7 : Bool;
      DiSpare8 : Bool;
      DiSpare9 : Bool;
      DiSpare10 : Bool;
   END_VAR
BEGIN
END_DATA_BLOCK

DATA_BLOCK "DiSimulation"   // DB103
{ S7_Optimized_Access := 'TRUE' }
// stored: AutoNumber false, MemoryReserve 100
   VAR
      ControlKey : Bool;
      EmergencyStop : Bool;
      CompressedAirPressureLow : Bool;
      PowerFailure : Bool;
      PowerReset : Bool;
      MagneticMixerFeedback : Bool;
      CipPumpFeedback : Bool;
      MagneticMixerOverload : Bool;
      CipPumpOverload : Bool;
      RuptureDisc : Bool;
      Cp01FlowSwitch : Bool;
      DiSpare1 : Bool;
      DiSpare2 : Bool;
      MMHighSpeedSensor : Bool;
      DiSpare3 : Bool;
      DiSpare4 : Bool;
      DiSpare5 : Bool;
      DiSpare6 : Bool;
      DiSpare7 : Bool;
      DiSpare8 : Bool;
      DiSpare9 : Bool;
      DiSpare10 : Bool;
   END_VAR
BEGIN
END_DATA_BLOCK

DATA_BLOCK "DoManualModeDb"   // DB2
{ S7_Optimized_Access := 'FALSE' }
// stored: AutoNumber false
   VAR
      Mm01Cmd : Bool;
      Cp01Cmd : Bool;
      Htr : Bool;
      Lf01 : Bool;
      DoSpare1 : Bool;
      DoSpare2 : Bool;
      DoSpare3 : Bool;
      DoSpare4 : Bool;
      DoSpare5 : Bool;
      DoSpare6 : Bool;
   END_VAR
BEGIN
END_DATA_BLOCK

ORGANIZATION_BLOCK "Main"   // OB1, LAD, ProgramCycle
TITLE = "Main Program Sweep (Cycle)"
{ S7_Optimized_Access := 'TRUE' }
// stored: SetENOAutomatically false
   VAR_INPUT
      Initial_Call : Bool;   // Initial call of this OB
      Remanence : Bool;   // =True, if remanent data are available
   END_VAR
   VAR_TEMP   // added for the SCL form of the ladder/FBD networks
      _w1 : Bool;
   END_VAR
BEGIN

REGION Network 1: "Sec_Pulse"
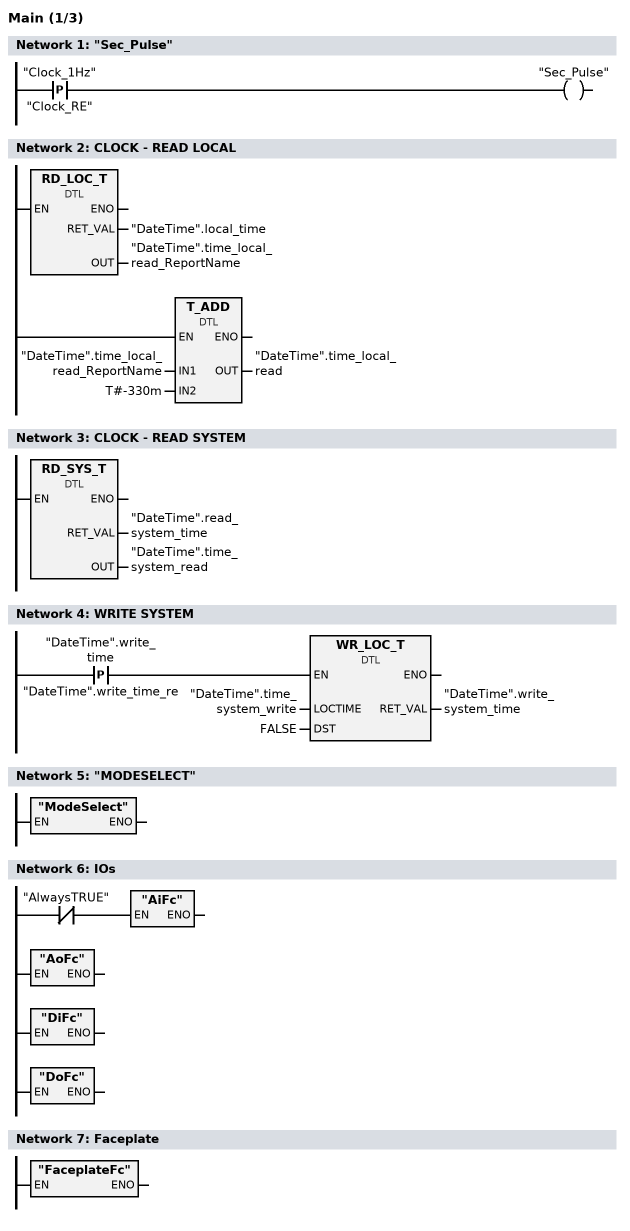
   RUNG wire#powerrail
      P_Contact(operand := "Clock_1Hz", bit := "Clock_RE")
      Coil( "Sec_Pulse" )
   END_RUNG
   // the same network as SCL:
   #_w1 := "Clock_1Hz" AND NOT "Clock_RE";   // rising edge of "Clock_1Hz"
   "Clock_RE" := "Clock_1Hz";
   "Sec_Pulse" := #_w1;
END_REGION

REGION Network 2: CLOCK - READ LOCAL
   RUNG wire#powerrail
      { S7_Templates := "date_type := DTL" } RD_LOC_T(RET_VAL => "DateTime".local_time, OUT => "DateTime".time_local_read_ReportName)
   END_RUNG
   RUNG wire#powerrail
      { S7_Templates := "[date_type := DTL, time_type := Time]" } T_ADD(IN1 := "DateTime".time_local_read_ReportName, IN2 := T#-330m, OUT => "DateTime".time_local_read)
   END_RUNG
   // the same network as SCL:
   "DateTime".local_time := RD_LOC_T(OUT => "DateTime".time_local_read_ReportName);
   T_ADD(IN1 := "DateTime".time_local_read_ReportName, IN2 := T#-330m, OUT => "DateTime".time_local_read);
END_REGION

REGION Network 3: CLOCK - READ SYSTEM
   RUNG wire#powerrail
      { S7_Templates := "date_type := DTL" } RD_SYS_T(RET_VAL => "DateTime".read_system_time, OUT => "DateTime".time_system_read)
   END_RUNG
   // the same network as SCL:
   "DateTime".read_system_time := RD_SYS_T(OUT => "DateTime".time_system_read);
END_REGION

REGION Network 4: WRITE SYSTEM
   RUNG wire#powerrail
      P_Contact(operand := "DateTime".write_time, bit := "DateTime".write_time_re)
      { S7_Templates := "loctime_type := DTL" } WR_LOC_T(LOCTIME := "DateTime".time_system_write, DST := FALSE, Ret_Val => "DateTime".write_system_time)
   END_RUNG
   // the same network as SCL:
   #_w1 := "DateTime".write_time AND NOT "DateTime".write_time_re;   // rising edge of "DateTime".write_time
   "DateTime".write_time_re := "DateTime".write_time;
   IF #_w1 THEN
       "DateTime".write_system_time := WR_LOC_T(LOCTIME := "DateTime".time_system_write, DST := FALSE);
   END_IF;
END_REGION

REGION Network 5: "MODESELECT"
   RUNG wire#powerrail
      "ModeSelect"()
   END_RUNG
   // the same network as SCL:
   "ModeSelect"();
END_REGION

REGION Network 6: IOs
   RUNG wire#powerrail
      I_Contact( "AlwaysTRUE" )
      "AiFc"()
   END_RUNG
   RUNG wire#powerrail
      "AoFc"()
   END_RUNG
   RUNG wire#powerrail
      "DiFc"()
   END_RUNG
   RUNG wire#powerrail
      "DoFc"()
   END_RUNG
   // the same network as SCL:
   IF NOT "AlwaysTRUE" THEN "AiFc"(); END_IF;
   "AoFc"();
   "DiFc"();
   "DoFc"();
END_REGION

REGION Network 7: Faceplate
   RUNG wire#powerrail
      "FaceplateFc"()
   END_RUNG
   // the same network as SCL:
   "FaceplateFc"();
END_REGION

REGION Network 8: ValvesOutputFc
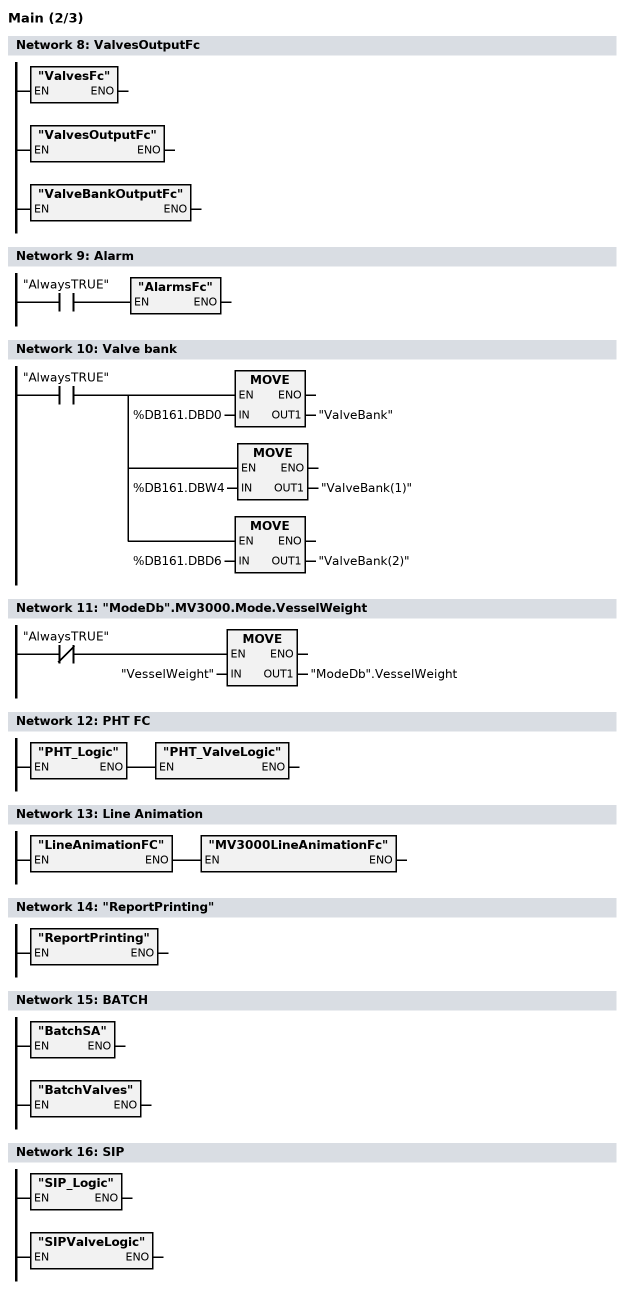
   RUNG wire#powerrail
      "ValvesFc"()
   END_RUNG
   RUNG wire#powerrail
      "ValvesOutputFc"()
   END_RUNG
   RUNG wire#powerrail
      "ValveBankOutputFc"()
   END_RUNG
   // the same network as SCL:
   "ValvesFc"();
   "ValvesOutputFc"();
   "ValveBankOutputFc"();
END_REGION

REGION Network 9: Alarm
   RUNG wire#powerrail
      Contact( "AlwaysTRUE" )
      "AlarmsFc"()
   END_RUNG
   // the same network as SCL:
   IF "AlwaysTRUE" THEN "AlarmsFc"(); END_IF;
END_REGION

REGION Network 10: Valve bank
   RUNG wire#powerrail
      Contact( "AlwaysTRUE" )
      wire#w1
      Move(in := %DB161.DBD0, out1 => "ValveBank")
   END_RUNG
   RUNG wire#w1
      Move(in := %DB161.DBW4, out1 => "ValveBank(1)")
   END_RUNG
   RUNG wire#w1
      Move(in := %DB161.DBD6, out1 => "ValveBank(2)")
   END_RUNG
   // the same network as SCL:
   IF "AlwaysTRUE" THEN
       "ValveBank" := %DB161.DBD0;
       "ValveBank(1)" := %DB161.DBW4;
       "ValveBank(2)" := %DB161.DBD6;
   END_IF;
END_REGION

REGION Network 11: "ModeDb".MV3000.Mode.VesselWeight
   RUNG wire#powerrail
      I_Contact( "AlwaysTRUE" )
      Move(in := "VesselWeight", out1 => "ModeDb".VesselWeight)
   END_RUNG
   // the same network as SCL:
   IF NOT "AlwaysTRUE" THEN "ModeDb".VesselWeight := "VesselWeight"; END_IF;
END_REGION

REGION Network 12: PHT FC
   RUNG wire#powerrail
      "PHT_Logic"()
      "PHT_ValveLogic"()
   END_RUNG
   // the same network as SCL:
   "PHT_Logic"(ENO => #_w1);
   IF #_w1 THEN "PHT_ValveLogic"(); END_IF;
END_REGION

REGION Network 13: Line Animation
   RUNG wire#powerrail
      "LineAnimationFC"()
      "MV3000LineAnimationFc"()
   END_RUNG
   // the same network as SCL:
   "LineAnimationFC"(ENO => #_w1);
   IF #_w1 THEN "MV3000LineAnimationFc"(); END_IF;
END_REGION

REGION Network 14: "ReportPrinting"
   RUNG wire#powerrail
      "ReportPrinting"()
   END_RUNG
   // the same network as SCL:
   "ReportPrinting"();
END_REGION

REGION Network 15: BATCH
   RUNG wire#powerrail
      "BatchSA"()
   END_RUNG
   RUNG wire#powerrail
      "BatchValves"()
   END_RUNG
   // the same network as SCL:
   "BatchSA"();
   "BatchValves"();
END_REGION

REGION Network 16: SIP
   RUNG wire#powerrail
      "SIP_Logic"()
   END_RUNG
   RUNG wire#powerrail
      "SIPValveLogic"()
   END_RUNG
   // the same network as SCL:
   "SIP_Logic"();
   "SIPValveLogic"();
END_REGION

REGION Network 17: CIP
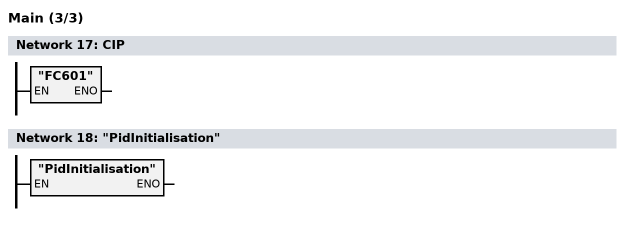
   RUNG wire#powerrail
      "FC601"()
   END_RUNG
   // the same network as SCL:
   "FC601"();
END_REGION

REGION Network 18: "PidInitialisation"
   RUNG wire#powerrail
      "PidInitialisation"()
   END_RUNG
   // the same network as SCL:
   "PidInitialisation"();
END_REGION
END_ORGANIZATION_BLOCK

FUNCTION "ModeSelect" : Void   // FC7, LAD
{ S7_Optimized_Access := 'TRUE' }
// stored: AutoNumber false, SetENOAutomatically false
BEGIN

REGION Network 1: ****************************MV3000_Enable *****************************
END_REGION

REGION Network 2: "ModeDb".MV3000.Mode.ManualMode.Enable
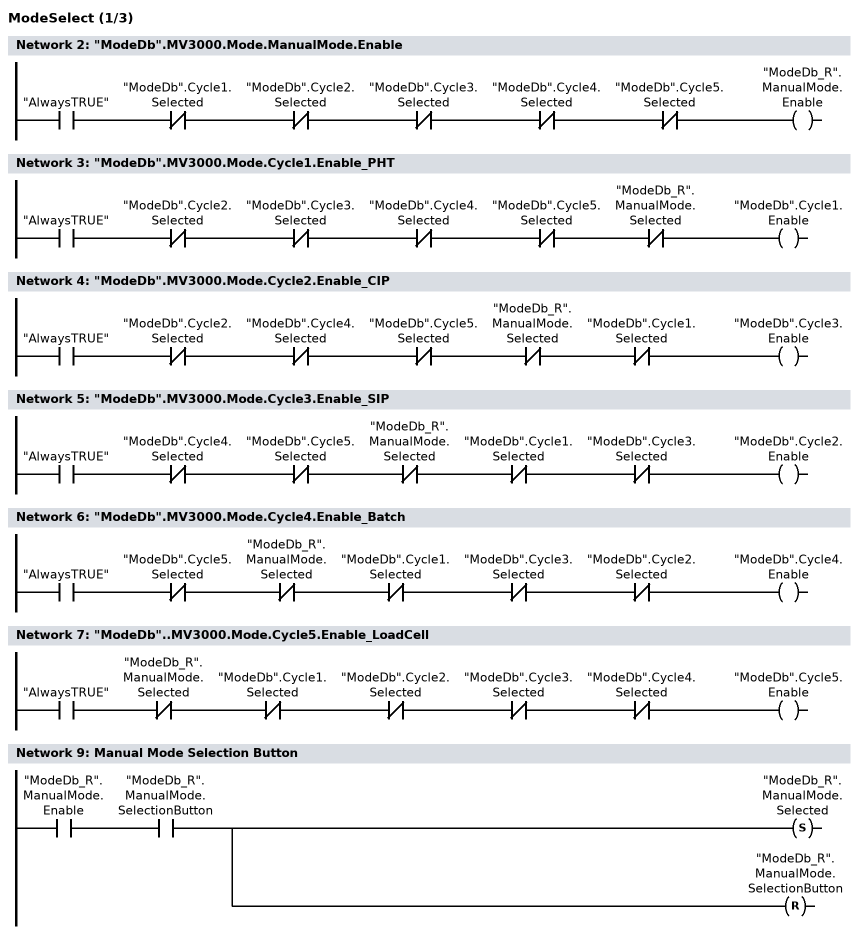
   RUNG wire#powerrail
      Contact( "AlwaysTRUE" )
      I_Contact( "ModeDb".Cycle1.Selected )
      I_Contact( "ModeDb".Cycle2.Selected )
      I_Contact( "ModeDb".Cycle3.Selected )
      I_Contact( "ModeDb".Cycle4.Selected )
      I_Contact( "ModeDb".Cycle5.Selected )
      Coil( "ModeDb_R".ManualMode.Enable )
   END_RUNG
   // the same network as SCL:
   "ModeDb_R".ManualMode.Enable := "AlwaysTRUE" AND NOT "ModeDb".Cycle1.Selected AND NOT "ModeDb".Cycle2.Selected AND NOT "ModeDb".Cycle3.Selected AND NOT "ModeDb".Cycle4.Selected AND NOT "ModeDb".Cycle5.Selected;
END_REGION

REGION Network 3: "ModeDb".MV3000.Mode.Cycle1.Enable_PHT
   RUNG wire#powerrail
      Contact( "AlwaysTRUE" )
      I_Contact( "ModeDb".Cycle2.Selected )
      I_Contact( "ModeDb".Cycle3.Selected )
      I_Contact( "ModeDb".Cycle4.Selected )
      I_Contact( "ModeDb".Cycle5.Selected )
      I_Contact( "ModeDb_R".ManualMode.Selected )
      Coil( "ModeDb".Cycle1.Enable )
   END_RUNG
   // the same network as SCL:
   "ModeDb".Cycle1.Enable := "AlwaysTRUE" AND NOT "ModeDb".Cycle2.Selected AND NOT "ModeDb".Cycle3.Selected AND NOT "ModeDb".Cycle4.Selected AND NOT "ModeDb".Cycle5.Selected AND NOT "ModeDb_R".ManualMode.Selected;
END_REGION

REGION Network 4: "ModeDb".MV3000.Mode.Cycle2.Enable_CIP
   RUNG wire#powerrail
      Contact( "AlwaysTRUE" )
      I_Contact( "ModeDb".Cycle2.Selected )
      I_Contact( "ModeDb".Cycle4.Selected )
      I_Contact( "ModeDb".Cycle5.Selected )
      I_Contact( "ModeDb_R".ManualMode.Selected )
      I_Contact( "ModeDb".Cycle1.Selected )
      Coil( "ModeDb".Cycle3.Enable )
   END_RUNG
   // the same network as SCL:
   "ModeDb".Cycle3.Enable := "AlwaysTRUE" AND NOT "ModeDb".Cycle2.Selected AND NOT "ModeDb".Cycle4.Selected AND NOT "ModeDb".Cycle5.Selected AND NOT "ModeDb_R".ManualMode.Selected AND NOT "ModeDb".Cycle1.Selected;
END_REGION

REGION Network 5: "ModeDb".MV3000.Mode.Cycle3.Enable_SIP
   RUNG wire#powerrail
      Contact( "AlwaysTRUE" )
      I_Contact( "ModeDb".Cycle4.Selected )
      I_Contact( "ModeDb".Cycle5.Selected )
      I_Contact( "ModeDb_R".ManualMode.Selected )
      I_Contact( "ModeDb".Cycle1.Selected )
      I_Contact( "ModeDb".Cycle3.Selected )
      Coil( "ModeDb".Cycle2.Enable )
   END_RUNG
   // the same network as SCL:
   "ModeDb".Cycle2.Enable := "AlwaysTRUE" AND NOT "ModeDb".Cycle4.Selected AND NOT "ModeDb".Cycle5.Selected AND NOT "ModeDb_R".ManualMode.Selected AND NOT "ModeDb".Cycle1.Selected AND NOT "ModeDb".Cycle3.Selected;
END_REGION

REGION Network 6: "ModeDb".MV3000.Mode.Cycle4.Enable_Batch
   RUNG wire#powerrail
      Contact( "AlwaysTRUE" )
      I_Contact( "ModeDb".Cycle5.Selected )
      I_Contact( "ModeDb_R".ManualMode.Selected )
      I_Contact( "ModeDb".Cycle1.Selected )
      I_Contact( "ModeDb".Cycle3.Selected )
      I_Contact( "ModeDb".Cycle2.Selected )
      Coil( "ModeDb".Cycle4.Enable )
   END_RUNG
   // the same network as SCL:
   "ModeDb".Cycle4.Enable := "AlwaysTRUE" AND NOT "ModeDb".Cycle5.Selected AND NOT "ModeDb_R".ManualMode.Selected AND NOT "ModeDb".Cycle1.Selected AND NOT "ModeDb".Cycle3.Selected AND NOT "ModeDb".Cycle2.Selected;
END_REGION

REGION Network 7: "ModeDb"..MV3000.Mode.Cycle5.Enable_LoadCell
   RUNG wire#powerrail
      Contact( "AlwaysTRUE" )
      I_Contact( "ModeDb_R".ManualMode.Selected )
      I_Contact( "ModeDb".Cycle1.Selected )
      I_Contact( "ModeDb".Cycle2.Selected )
      I_Contact( "ModeDb".Cycle3.Selected )
      I_Contact( "ModeDb".Cycle4.Selected )
      Coil( "ModeDb".Cycle5.Enable )
   END_RUNG
   // the same network as SCL:
   "ModeDb".Cycle5.Enable := "AlwaysTRUE" AND NOT "ModeDb_R".ManualMode.Selected AND NOT "ModeDb".Cycle1.Selected AND NOT "ModeDb".Cycle2.Selected AND NOT "ModeDb".Cycle3.Selected AND NOT "ModeDb".Cycle4.Selected;
END_REGION

REGION Network 8: ------------------------------------------------- SELECTION BUTTON -------------------------------------------------
END_REGION

REGION Network 9: Manual Mode Selection Button
   RUNG wire#powerrail
      Contact( "ModeDb_R".ManualMode.Enable )
      Contact( "ModeDb_R".ManualMode.SelectionButton )
      wire#w1
      S_Coil( "ModeDb_R".ManualMode.Selected )
   END_RUNG
   RUNG wire#w1
      R_Coil( "ModeDb_R".ManualMode.SelectionButton )
   END_RUNG
   // the same network as SCL:
   IF "ModeDb_R".ManualMode.Enable AND "ModeDb_R".ManualMode.SelectionButton THEN
       "ModeDb_R".ManualMode.Selected := TRUE;
       "ModeDb_R".ManualMode.SelectionButton := FALSE;
   END_IF;
END_REGION

REGION Network 10: __________________________ VESSEL STATUS__________________________
END_REGION

REGION Network 11: "HmiTags".Cv200VesselStatus
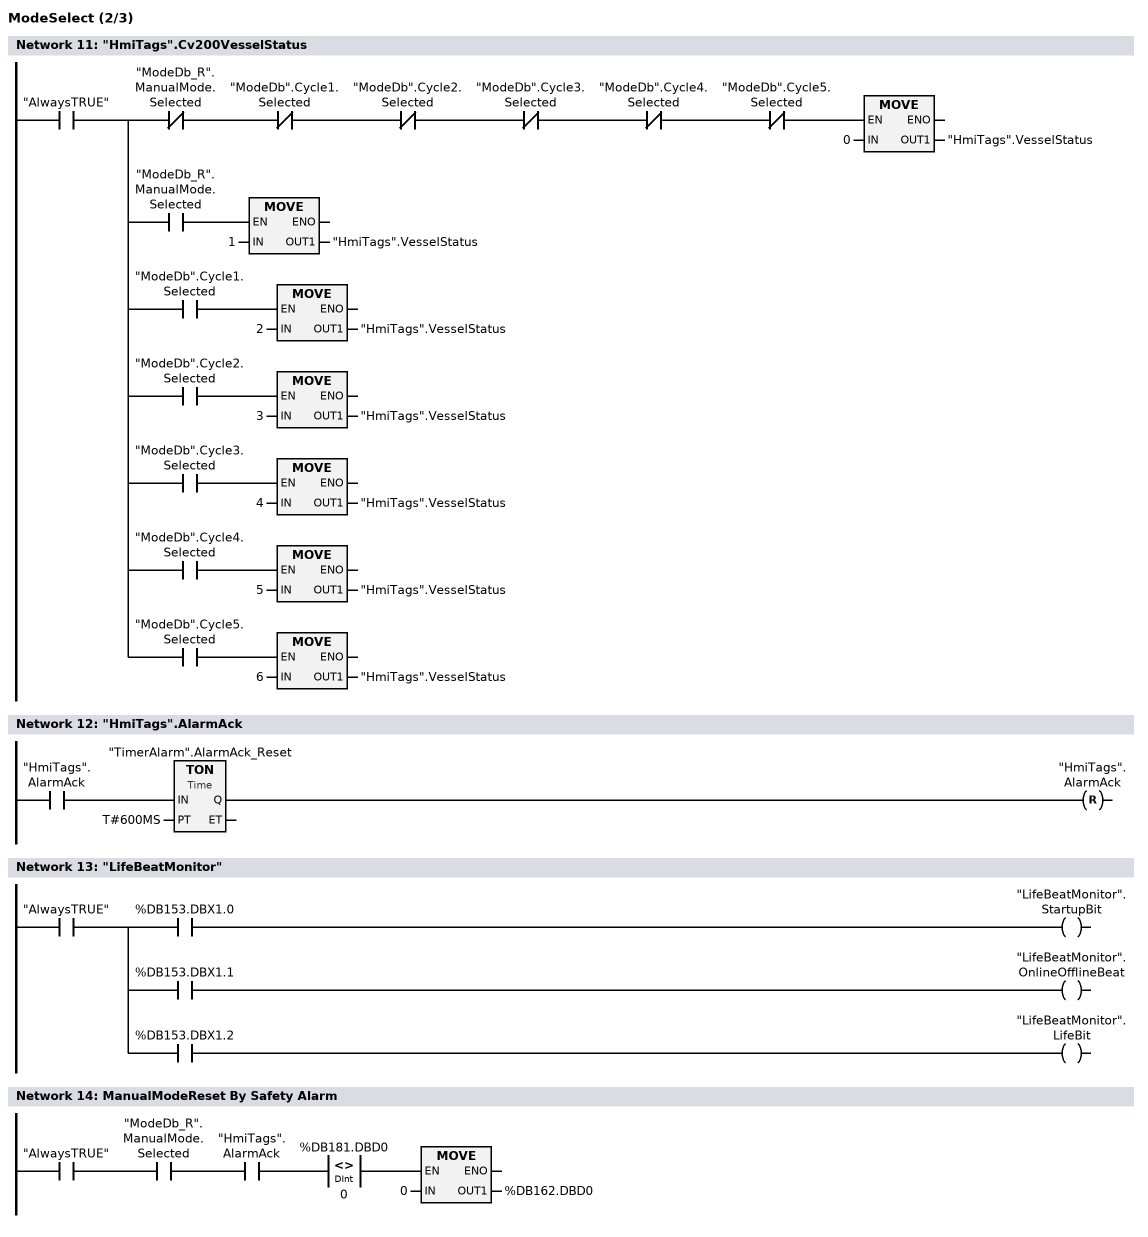
   RUNG wire#powerrail
      Contact( "AlwaysTRUE" )
      wire#w1
      I_Contact( "ModeDb_R".ManualMode.Selected )
      I_Contact( "ModeDb".Cycle1.Selected )
      I_Contact( "ModeDb".Cycle2.Selected )
      I_Contact( "ModeDb".Cycle3.Selected )
      I_Contact( "ModeDb".Cycle4.Selected )
      I_Contact( "ModeDb".Cycle5.Selected )
      Move(in := 0, out1 => "HmiTags".VesselStatus)
   END_RUNG
   RUNG wire#w1
      Contact( "ModeDb_R".ManualMode.Selected )
      Move(in := 1, out1 => "HmiTags".VesselStatus)
   END_RUNG
   RUNG wire#w1
      Contact( "ModeDb".Cycle1.Selected )
      Move(in := 2, out1 => "HmiTags".VesselStatus)
   END_RUNG
   RUNG wire#w1
      Contact( "ModeDb".Cycle2.Selected )
      Move(in := 3, out1 => "HmiTags".VesselStatus)
   END_RUNG
   RUNG wire#w1
      Contact( "ModeDb".Cycle3.Selected )
      Move(in := 4, out1 => "HmiTags".VesselStatus)
   END_RUNG
   RUNG wire#w1
      Contact( "ModeDb".Cycle4.Selected )
      Move(in := 5, out1 => "HmiTags".VesselStatus)
   END_RUNG
   RUNG wire#w1
      Contact( "ModeDb".Cycle5.Selected )
      Move(in := 6, out1 => "HmiTags".VesselStatus)
   END_RUNG
   // the same network as SCL:
   IF "AlwaysTRUE" AND NOT "ModeDb_R".ManualMode.Selected AND NOT "ModeDb".Cycle1.Selected AND NOT "ModeDb".Cycle2.Selected AND NOT "ModeDb".Cycle3.Selected AND NOT "ModeDb".Cycle4.Selected AND NOT "ModeDb".Cycle5.Selected THEN
       "HmiTags".VesselStatus := 0;
   END_IF;
   IF "AlwaysTRUE" AND "ModeDb_R".ManualMode.Selected THEN "HmiTags".VesselStatus := 1; END_IF;
   IF "AlwaysTRUE" AND "ModeDb".Cycle1.Selected THEN "HmiTags".VesselStatus := 2; END_IF;
   IF "AlwaysTRUE" AND "ModeDb".Cycle2.Selected THEN "HmiTags".VesselStatus := 3; END_IF;
   IF "AlwaysTRUE" AND "ModeDb".Cycle3.Selected THEN "HmiTags".VesselStatus := 4; END_IF;
   IF "AlwaysTRUE" AND "ModeDb".Cycle4.Selected THEN "HmiTags".VesselStatus := 5; END_IF;
   IF "AlwaysTRUE" AND "ModeDb".Cycle5.Selected THEN "HmiTags".VesselStatus := 6; END_IF;
END_REGION

REGION Network 12: "HmiTags".AlarmAck
   RUNG wire#powerrail
      Contact( "HmiTags".AlarmAck )
      { S7_Templates := "time_type := Time" } "TimerAlarm".AlarmAck_Reset.TON(pt := T#600MS, et =>)
      R_Coil( "HmiTags".AlarmAck )
   END_RUNG
   // the same network as SCL:
   "TimerAlarm".AlarmAck_Reset.TON(IN := "HmiTags".AlarmAck, PT := T#600MS);
   IF "TimerAlarm".AlarmAck_Reset.Q THEN "HmiTags".AlarmAck := FALSE; END_IF;
END_REGION

REGION Network 13: "LifeBeatMonitor"
   RUNG wire#powerrail
      Contact( "AlwaysTRUE" )
      wire#w1
      Contact( %DB153.DBX1.0 )
      Coil( "LifeBeatMonitor".StartupBit )
   END_RUNG
   RUNG wire#w1
      Contact( %DB153.DBX1.1 )
      Coil( "LifeBeatMonitor".OnlineOfflineBeat )
   END_RUNG
   RUNG wire#w1
      Contact( %DB153.DBX1.2 )
      Coil( "LifeBeatMonitor".LifeBit )
   END_RUNG
   // the same network as SCL:
   "LifeBeatMonitor".StartupBit := "AlwaysTRUE" AND %DB153.DBX1.0;
   "LifeBeatMonitor".OnlineOfflineBeat := "AlwaysTRUE" AND %DB153.DBX1.1;
   "LifeBeatMonitor".LifeBit := "AlwaysTRUE" AND %DB153.DBX1.2;
END_REGION

REGION Network 14: ManualModeReset By Safety Alarm
   RUNG wire#powerrail
      Contact( "AlwaysTRUE" )
      Contact( "ModeDb_R".ManualMode.Selected )
      Contact( "HmiTags".AlarmAck )
      { S7_Templates := "SrcType := DInt" } NE_Contact(in1 := %DB181.DBD0, in2 := 0)
      Move(in := 0, out1 => %DB162.DBD0)
   END_RUNG
   // the same network as SCL:
   IF "AlwaysTRUE" AND "ModeDb_R".ManualMode.Selected AND "HmiTags".AlarmAck AND (%DB181.DBD0 <> 0) THEN
       %DB162.DBD0 := 0;
   END_IF;
END_REGION

REGION Network 15: Master Reset
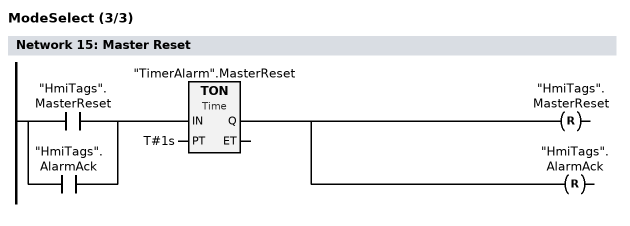
   RUNG wire#powerrail
      Contact( "HmiTags".MasterReset )
      wire#w1
      { S7_Templates := "time_type := Time" } "TimerAlarm".MasterReset.TON(pt := T#1s, et =>)
      wire#w2
      R_Coil( "HmiTags".MasterReset )
   END_RUNG
   RUNG wire#powerrail
      Contact( "HmiTags".AlarmAck )
   END_RUNG wire#w1
   RUNG wire#w2
      R_Coil( "HmiTags".AlarmAck )
   END_RUNG
   // the same network as SCL:
   "TimerAlarm".MasterReset.TON(IN := "HmiTags".MasterReset OR "HmiTags".AlarmAck, PT := T#1s);
   IF "TimerAlarm".MasterReset.Q THEN
       "HmiTags".MasterReset := FALSE;
       "HmiTags".AlarmAck := FALSE;
   END_IF;
END_REGION

REGION Network 16 (SCL): __________________________ Manual Mode Valve REset__________________________
   IF ("ModeDb_R".ManualMode.Abort  = 1 OR "HmiTags".MasterReset = 1) AND "ModeDb_R".ManualMode.Selected = 1 AND
       "ValveDb".Cv01.OpenClose =0 AND
       "ValveDb".Cv02.OpenClose =0 AND
       "ValveDb".Cv03.OpenClose=0  AND
       "ValveDb".Cv04.OpenClose=0 AND
       "ValveDb".Cv05.OpenClose=0 AND
       "ValveDb".Cv06.OpenClose=0 AND
       "ValveDb".Cv07.OpenClose=0 AND
       "ValveDb".Cv08.OpenClose=0 AND
       "ValveDb".Cv09.OpenClose=0 AND
       "ValveDb".Cv10.OpenClose=0 AND
       "ValveDb".Cv11.OpenClose=0 AND
       "ValveDb".Cv12.OpenClose=0 AND
       "ValveDb".Cv13.OpenClose=0 AND
       "ValveDb".Cv14.OpenClose=0 AND
       "ValveDb".Cv15.OpenClose=0 AND
       "ValveDb".Cv16.OpenClose=0 AND
       "ValveDb".Cv17.OpenClose=0 AND
       "ValveDb".Cv18.OpenClose=0 AND
       "ValveDb".Cv19.OpenClose=0 AND
       "ValveDb".Cv20.OpenClose=0 AND
       "ValveDb".Cv21.OpenClose=0 AND
       "ValveDb".Cv22.OpenClose=0 AND
       "ValveDb".Cv23.OpenClose=0 AND
       "ValveDb".Cv24.OpenClose=0 AND
       "ValveDb".Cv25.OpenClose=0 AND
       "ValveDb".Cv26.OpenClose=0 AND
       "ValveDb".Cv27.OpenClose=0 AND
       "ValveDb".Cv28.OpenClose=0 AND
       "ValveDb".Cv29.OpenClose=0 AND
       "ValveDb".Cv30.OpenClose=0 AND
       "ValveDb".Cv31.OpenClose=0 AND
       "ValveDb".Cv32.OpenClose=0 AND
       "ValveDb".Cv33.OpenClose=0 AND
       "ValveDb".Cv34.OpenClose=0 AND
       "ValveDb".Cv35.OpenClose=0 AND
       "ValveDb".Cv36.OpenClose=0 AND
       "ValveDb".Cv37.OpenClose=0 AND
       "ValveDb".Cv38.OpenClose=0 AND
       "ValveDb".Cv39.OpenClose=0 AND  
       "ValveDb".Cv40.OpenClose=0 AND
       "ValveDb".Cv41.OpenClose=0 AND
       "ValveDb".Cv42.OpenClose=0 AND
       "ValveDb".Cv43.OpenClose=0 AND
       "ValveDb".Cv44.OpenClose=0 AND
       "ValveDb".Cv45.OpenClose=0 AND
       "ValveDb".Cv46.OpenClose=0 AND
       "ValveDb".Cv47.OpenClose=0 AND
       "ValveDb".Cv48.OpenClose=0 AND
       "ValveDb".Cv49.OpenClose=0 AND
       "ValveDb".Cv50.OpenClose=0 AND
       "ValveDb".Cv51.OpenClose=0 AND
       "ValveDb".Cv52.OpenClose=0 AND
       "ValveDb".Cv53.OpenClose=0 AND
       "ValveDb".Cv54.OpenClose=0 AND
       "ValveDb".Cv55.OpenClose=0 AND
       "ValveDb".Cv56.OpenClose=0 AND
       "ValveDb".Cv57.OpenClose=0 AND
       "ValveDb".Cv58.OpenClose=0 AND
       "ValveDb".Cv59.OpenClose=0 AND
       "ValveDb".Cv60.OpenClose=0 AND
       "ValveDb".Cv61.OpenClose=0 AND
       "ValveDb".Cv62.OpenClose=0 AND
       "ValveDb".Cv63.OpenClose=0 AND
       "ValveDb".Cv64.OpenClose=0 AND
       "ValveDb".Fbov01.OpenClose=0




   THEN
       "ModeDb_R".ManualMode.Selected := 0 ;
   END_IF;
END_REGION
END_FUNCTION

FUNCTION "AiFc" : Void   // FC108, LAD
{ S7_Optimized_Access := 'TRUE' }
// stored: AutoNumber false, SetENOAutomatically false
BEGIN

REGION Network 1: "AiDb"
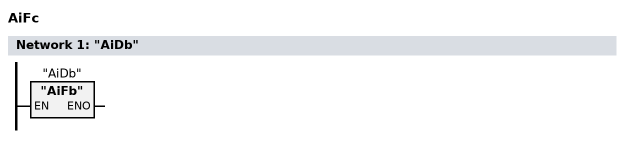
   RUNG wire#powerrail
      "AiDb"()
   END_RUNG
   // the same network as SCL:
   "AiDb"();   // "AiFb"
END_REGION

REGION Network 2 (SCL): AnalogInputIw
   "AiDb".Ai01.AnalogInputIw := "Ticr01NfcoLineTemp";
   "AiDb".Ai02.AnalogInputIw := "Ticr02VfcoLineTemp";
   "AiDb".Ai03.AnalogInputIw := "AiSpare01";
   "AiDb".Ai04.AnalogInputIw := "AiSpare02";
   "AiDb".Ai05.AnalogInputIw := "AiSpare03";
   "AiDb".Ai06.AnalogInputIw := "Ticr06Pf01InLineTemp";
   "AiDb".Ai07.AnalogInputIw := "Ticr07Pf02InLineTemp";
   "AiDb".Ai08.AnalogInputIw := "Ticr08Pf02OutLineTemp";
   "AiDb".Ai09.AnalogInputIw := "Ticr09PtlDrainTemp";
   "AiDb".Ai10.AnalogInputIw := "Ticr10VesselTemp";
   "AiDb".Ai11.AnalogInputIw := "Picr01VesselPressure";
   "AiDb".Ai12.AnalogInputIw := "Picr02VesselRclLine";
   "AiDb".Ai13.AnalogInputIw := "Picr03Pf01OutLinePressure";
   "AiDb".Ai14.AnalogInputIw := "Picr04Pf02OutLinePressure";
   "AiDb".Ai15.AnalogInputIw := "Cicr01ProcessDrainConductivity";
   "AiDb".Ai16.AnalogInputIw := "AiSpare04";
   "AiDb".Ai17.AnalogInputIw := "AiSpare05";
   "AiDb".Ai18.AnalogInputIw := "AiSpare06";
   "AiDb".Ai19.AnalogInputIw := "AiSpare07";
   "AiDb".Ai20.AnalogInputIw := "AiSpare08";
   "AiDb".Ai21.AnalogInputIw := "AiSpare09";
   "AiDb".Ai22.AnalogInputIw := "AiSpare10";
   "AiDb".Ai23.AnalogInputIw := "AiSpare11";
   "AiDb".Ai24.AnalogInputIw := "AiSpare12";
END_REGION
END_FUNCTION

FUNCTION_BLOCK "AiFb"   // FB108, LAD
{ S7_Optimized_Access := 'TRUE' }
// stored: AutoNumber false, MemoryReserve 100, SetENOAutomatically false
   VAR
      Ai01 { S7_SetPoint := 'True'} : "FB:Analog_Scaling";   // NfcoLineTemp(Ticr01)
      Ai02 { S7_SetPoint := 'True'} : "FB:Analog_Scaling";   // VfcoLineTemp(Ticr02)
      Ai03 { S7_SetPoint := 'True'} : "FB:Analog_Scaling";   // AiSpare01
      Ai04 { S7_SetPoint := 'True'} : "FB:Analog_Scaling";   // AiSpare02
      Ai05 { S7_SetPoint := 'True'} : "FB:Analog_Scaling";   // AiSpare03
      Ai06 { S7_SetPoint := 'True'} : "FB:Analog_Scaling";   // Pf01InLineTemp(Ticr06)
      Ai07 { S7_SetPoint := 'True'} : "FB:Analog_Scaling";   // Pf02InLineTemp(Ticr07)
      Ai08 { S7_SetPoint := 'True'} : "FB:Analog_Scaling";   // Pf02OutLineTemp(Ticr08)
      Ai09 { S7_SetPoint := 'True'} : "FB:Analog_Scaling";   // PtlDrainTemp(Ticr09)
      Ai10 { S7_SetPoint := 'True'} : "FB:Analog_Scaling";   // VesselTemp(Ticr10)
      Ai11 { S7_SetPoint := 'True'} : "FB:Analog_Scaling";   // VesselPressure(Picr01)
      Ai12 { S7_SetPoint := 'True'} : "FB:Analog_Scaling";   // VesselRclLine(Picr02)
      Ai13 { S7_SetPoint := 'True'} : "FB:Analog_Scaling";   // Pf01OutLinePressure(Picr03)
      Ai14 { S7_SetPoint := 'True'} : "FB:Analog_Scaling";   // Pf02OutLinePressure(Picr04)
      Ai15 { S7_SetPoint := 'True'} : "FB:Analog_Scaling";   // ProcessDrainConductivity
      Ai16 { S7_SetPoint := 'True'} : "FB:Analog_Scaling";   // AiSpare04
      Ai17 { S7_SetPoint := 'True'} : "FB:Analog_Scaling";   // AiSpare05
      Ai18 { S7_SetPoint := 'True'} : "FB:Analog_Scaling";   // AiSpare06
      Ai19 { S7_SetPoint := 'True'} : "FB:Analog_Scaling";   // AiSpare07
      Ai20 { S7_SetPoint := 'True'} : "FB:Analog_Scaling";   // AiSpare08
      Ai21 { S7_SetPoint := 'True'} : "FB:Analog_Scaling";   // AiSpare09
      Ai22 { S7_SetPoint := 'True'} : "FB:Analog_Scaling";   // AiSpare10
      Ai23 { S7_SetPoint := 'True'} : "FB:Analog_Scaling";   // AiSpare11
      Ai24 { S7_SetPoint := 'True'} : "FB:Analog_Scaling";   // AiSpare12
   END_VAR
BEGIN

REGION Network 1: #Ai01--- NfcoLineTemp
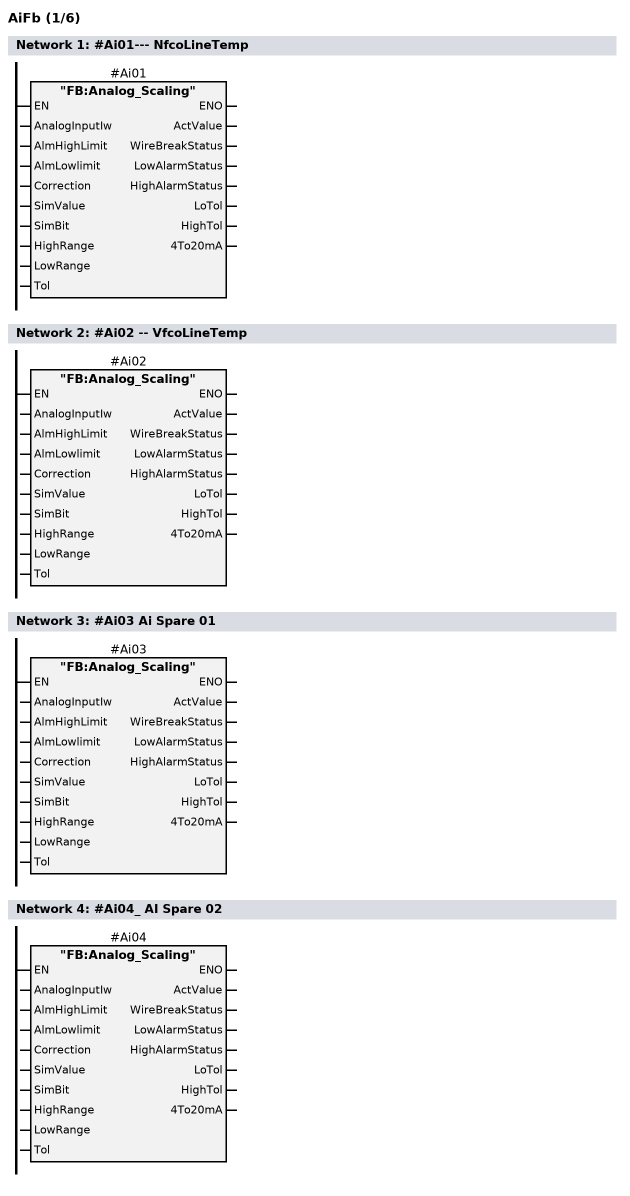
   RUNG wire#powerrail
      #Ai01(AnalogInputIw :=, AlmHighLimit :=, AlmLowlimit :=, Correction :=, SimValue :=, SimBit :=, HighRange :=, LowRange :=, Tol :=, ActValue =>, WireBreakStatus =>, LowAlarmStatus =>, HighAlarmStatus =>, LoTol =>, HighTol =>, "4To20mA" =>)
   END_RUNG
   // the same network as SCL:
   #Ai01();   // "FB:Analog_Scaling"
END_REGION

REGION Network 2: #Ai02 -- VfcoLineTemp
   RUNG wire#powerrail
      #Ai02(AnalogInputIw :=, AlmHighLimit :=, AlmLowlimit :=, Correction :=, SimValue :=, SimBit :=, HighRange :=, LowRange :=, Tol :=, ActValue =>, WireBreakStatus =>, LowAlarmStatus =>, HighAlarmStatus =>, LoTol =>, HighTol =>, "4To20mA" =>)
   END_RUNG
   // the same network as SCL:
   #Ai02();   // "FB:Analog_Scaling"
END_REGION

REGION Network 3: #Ai03 Ai Spare 01
   RUNG wire#powerrail
      #Ai03(AnalogInputIw :=, AlmHighLimit :=, AlmLowlimit :=, Correction :=, SimValue :=, SimBit :=, HighRange :=, LowRange :=, Tol :=, ActValue =>, WireBreakStatus =>, LowAlarmStatus =>, HighAlarmStatus =>, LoTol =>, HighTol =>, "4To20mA" =>)
   END_RUNG
   // the same network as SCL:
   #Ai03();   // "FB:Analog_Scaling"
END_REGION

REGION Network 4: #Ai04_ AI Spare 02
   RUNG wire#powerrail
      #Ai04(AnalogInputIw :=, AlmHighLimit :=, AlmLowlimit :=, Correction :=, SimValue :=, SimBit :=, HighRange :=, LowRange :=, Tol :=, ActValue =>, WireBreakStatus =>, LowAlarmStatus =>, HighAlarmStatus =>, LoTol =>, HighTol =>, "4To20mA" =>)
   END_RUNG
   // the same network as SCL:
   #Ai04();   // "FB:Analog_Scaling"
END_REGION

REGION Network 5: #Ai05--- #Ai04_ AI Spare 03
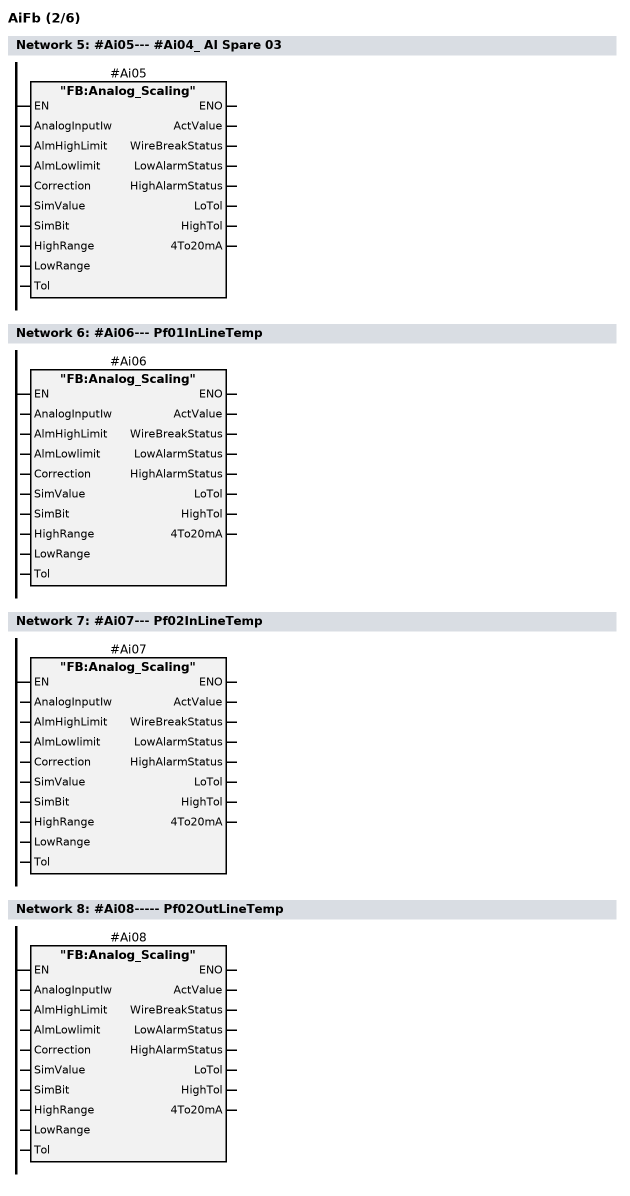
   RUNG wire#powerrail
      #Ai05(AnalogInputIw :=, AlmHighLimit :=, AlmLowlimit :=, Correction :=, SimValue :=, SimBit :=, HighRange :=, LowRange :=, Tol :=, ActValue =>, WireBreakStatus =>, LowAlarmStatus =>, HighAlarmStatus =>, LoTol =>, HighTol =>, "4To20mA" =>)
   END_RUNG
   // the same network as SCL:
   #Ai05();   // "FB:Analog_Scaling"
END_REGION

REGION Network 6: #Ai06--- Pf01InLineTemp
   RUNG wire#powerrail
      #Ai06(AnalogInputIw :=, AlmHighLimit :=, AlmLowlimit :=, Correction :=, SimValue :=, SimBit :=, HighRange :=, LowRange :=, Tol :=, ActValue =>, WireBreakStatus =>, LowAlarmStatus =>, HighAlarmStatus =>, LoTol =>, HighTol =>, "4To20mA" =>)
   END_RUNG
   // the same network as SCL:
   #Ai06();   // "FB:Analog_Scaling"
END_REGION

REGION Network 7: #Ai07--- Pf02InLineTemp
   RUNG wire#powerrail
      #Ai07(AnalogInputIw :=, AlmHighLimit :=, AlmLowlimit :=, Correction :=, SimValue :=, SimBit :=, HighRange :=, LowRange :=, Tol :=, ActValue =>, WireBreakStatus =>, LowAlarmStatus =>, HighAlarmStatus =>, LoTol =>, HighTol =>, "4To20mA" =>)
   END_RUNG
   // the same network as SCL:
   #Ai07();   // "FB:Analog_Scaling"
END_REGION

REGION Network 8: #Ai08----- Pf02OutLineTemp
   RUNG wire#powerrail
      #Ai08(AnalogInputIw :=, AlmHighLimit :=, AlmLowlimit :=, Correction :=, SimValue :=, SimBit :=, HighRange :=, LowRange :=, Tol :=, ActValue =>, WireBreakStatus =>, LowAlarmStatus =>, HighAlarmStatus =>, LoTol =>, HighTol =>, "4To20mA" =>)
   END_RUNG
   // the same network as SCL:
   #Ai08();   // "FB:Analog_Scaling"
END_REGION

REGION Network 9: #Ai09---- PtlDrainTemp
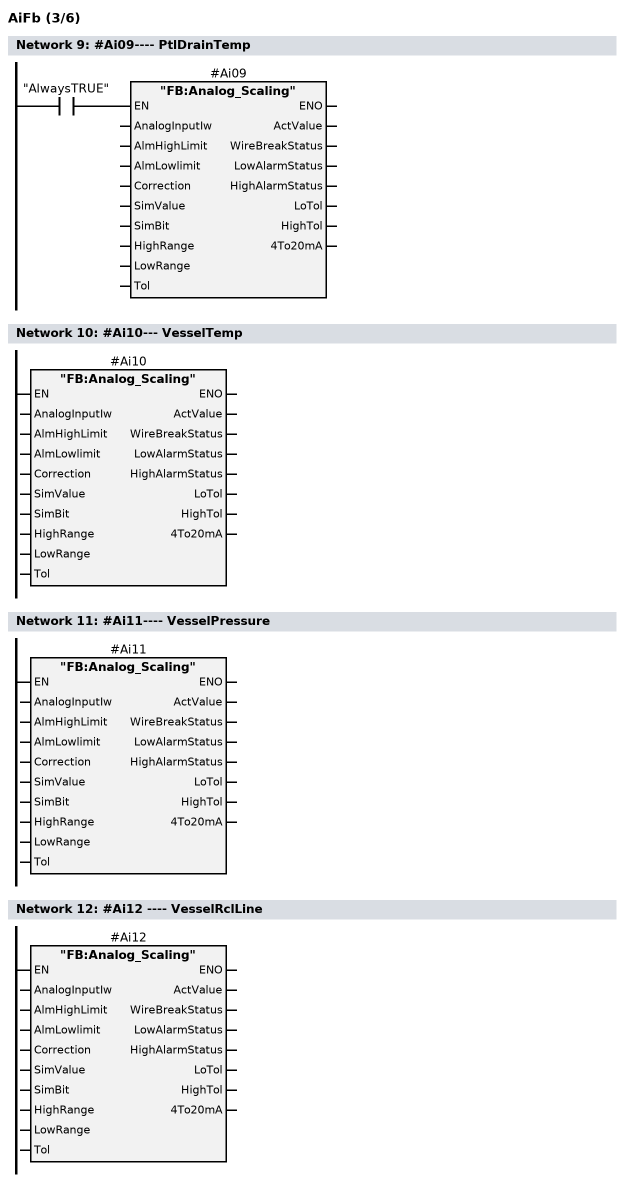
   RUNG wire#powerrail
      Contact( "AlwaysTRUE" )
      #Ai09(AnalogInputIw :=, AlmHighLimit :=, AlmLowlimit :=, Correction :=, SimValue :=, SimBit :=, HighRange :=, LowRange :=, Tol :=, ActValue =>, WireBreakStatus =>, LowAlarmStatus =>, HighAlarmStatus =>, LoTol =>, HighTol =>, "4To20mA" =>)
   END_RUNG
   // the same network as SCL:
   IF "AlwaysTRUE" THEN
       #Ai09();   // "FB:Analog_Scaling"
   END_IF;
END_REGION

REGION Network 10: #Ai10--- VesselTemp
   RUNG wire#powerrail
      #Ai10(AnalogInputIw :=, AlmHighLimit :=, AlmLowlimit :=, Correction :=, SimValue :=, SimBit :=, HighRange :=, LowRange :=, Tol :=, ActValue =>, WireBreakStatus =>, LowAlarmStatus =>, HighAlarmStatus =>, LoTol =>, HighTol =>, "4To20mA" =>)
   END_RUNG
   // the same network as SCL:
   #Ai10();   // "FB:Analog_Scaling"
END_REGION

REGION Network 11: #Ai11---- VesselPressure
   RUNG wire#powerrail
      #Ai11(AnalogInputIw :=, AlmHighLimit :=, AlmLowlimit :=, Correction :=, SimValue :=, SimBit :=, HighRange :=, LowRange :=, Tol :=, ActValue =>, WireBreakStatus =>, LowAlarmStatus =>, HighAlarmStatus =>, LoTol =>, HighTol =>, "4To20mA" =>)
   END_RUNG
   // the same network as SCL:
   #Ai11();   // "FB:Analog_Scaling"
END_REGION

REGION Network 12: #Ai12 ---- VesselRclLine
   RUNG wire#powerrail
      #Ai12(AnalogInputIw :=, AlmHighLimit :=, AlmLowlimit :=, Correction :=, SimValue :=, SimBit :=, HighRange :=, LowRange :=, Tol :=, ActValue =>, WireBreakStatus =>, LowAlarmStatus =>, HighAlarmStatus =>, LoTol =>, HighTol =>, "4To20mA" =>)
   END_RUNG
   // the same network as SCL:
   #Ai12();   // "FB:Analog_Scaling"
END_REGION

REGION Network 13: #Ai13--- Pf01OutLinePressure
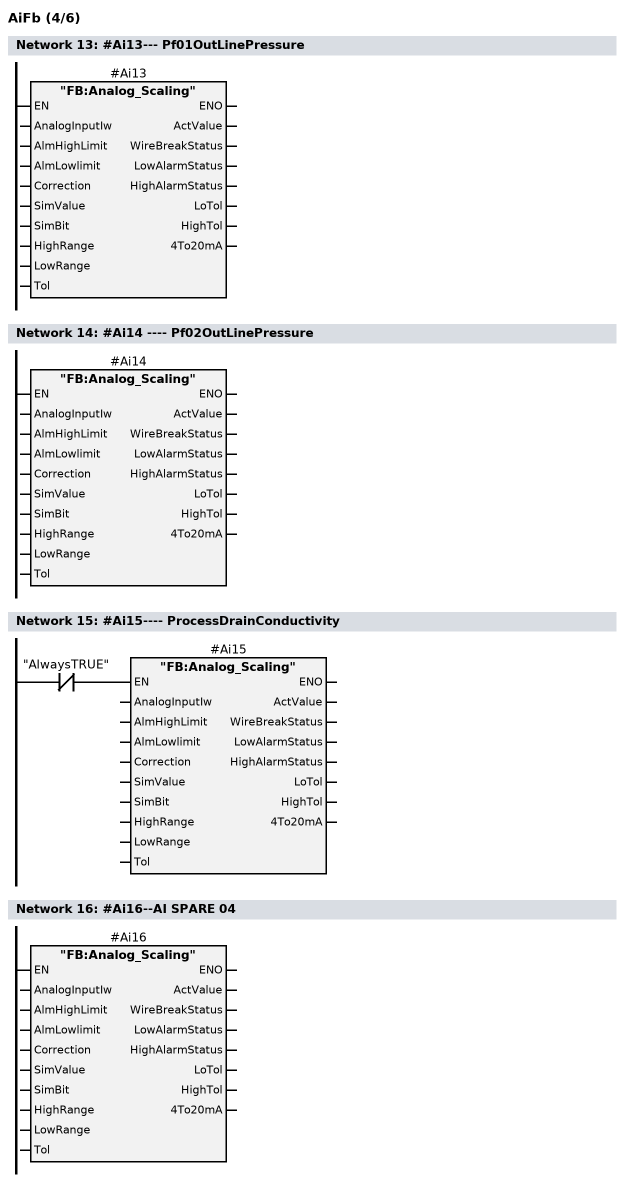
   RUNG wire#powerrail
      #Ai13(AnalogInputIw :=, AlmHighLimit :=, AlmLowlimit :=, Correction :=, SimValue :=, SimBit :=, HighRange :=, LowRange :=, Tol :=, ActValue =>, WireBreakStatus =>, LowAlarmStatus =>, HighAlarmStatus =>, LoTol =>, HighTol =>, "4To20mA" =>)
   END_RUNG
   // the same network as SCL:
   #Ai13();   // "FB:Analog_Scaling"
END_REGION

REGION Network 14: #Ai14 ---- Pf02OutLinePressure
   RUNG wire#powerrail
      #Ai14(AnalogInputIw :=, AlmHighLimit :=, AlmLowlimit :=, Correction :=, SimValue :=, SimBit :=, HighRange :=, LowRange :=, Tol :=, ActValue =>, WireBreakStatus =>, LowAlarmStatus =>, HighAlarmStatus =>, LoTol =>, HighTol =>, "4To20mA" =>)
   END_RUNG
   // the same network as SCL:
   #Ai14();   // "FB:Analog_Scaling"
END_REGION

REGION Network 15: #Ai15---- ProcessDrainConductivity
   RUNG wire#powerrail
      I_Contact( "AlwaysTRUE" )
      #Ai15(AnalogInputIw :=, AlmHighLimit :=, AlmLowlimit :=, Correction :=, SimValue :=, SimBit :=, HighRange :=, LowRange :=, Tol :=, ActValue =>, WireBreakStatus =>, LowAlarmStatus =>, HighAlarmStatus =>, LoTol =>, HighTol =>, "4To20mA" =>)
   END_RUNG
   // the same network as SCL:
   IF NOT "AlwaysTRUE" THEN
       #Ai15();   // "FB:Analog_Scaling"
   END_IF;
END_REGION

REGION Network 16: #Ai16--AI SPARE 04
   RUNG wire#powerrail
      #Ai16(AnalogInputIw :=, AlmHighLimit :=, AlmLowlimit :=, Correction :=, SimValue :=, SimBit :=, HighRange :=, LowRange :=, Tol :=, ActValue =>, WireBreakStatus =>, LowAlarmStatus =>, HighAlarmStatus =>, LoTol =>, HighTol =>, "4To20mA" =>)
   END_RUNG
   // the same network as SCL:
   #Ai16();   // "FB:Analog_Scaling"
END_REGION

REGION Network 17: #Ai17--AI SPARE 05
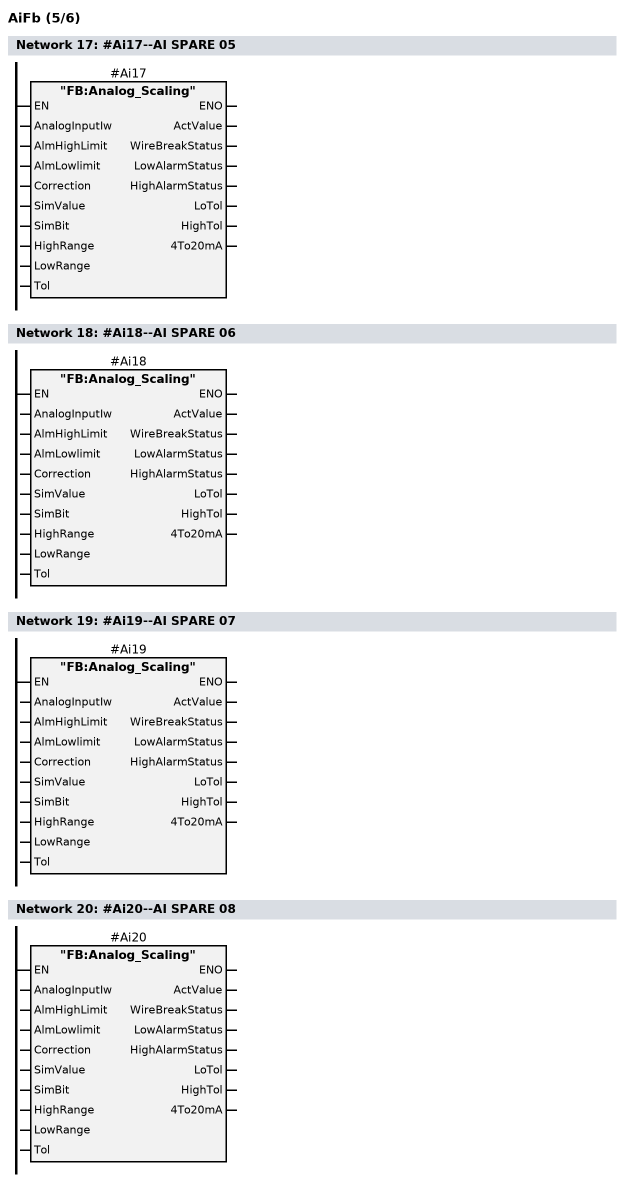
   RUNG wire#powerrail
      #Ai17(AnalogInputIw :=, AlmHighLimit :=, AlmLowlimit :=, Correction :=, SimValue :=, SimBit :=, HighRange :=, LowRange :=, Tol :=, ActValue =>, WireBreakStatus =>, LowAlarmStatus =>, HighAlarmStatus =>, LoTol =>, HighTol =>, "4To20mA" =>)
   END_RUNG
   // the same network as SCL:
   #Ai17();   // "FB:Analog_Scaling"
END_REGION

REGION Network 18: #Ai18--AI SPARE 06
   RUNG wire#powerrail
      #Ai18(AnalogInputIw :=, AlmHighLimit :=, AlmLowlimit :=, Correction :=, SimValue :=, SimBit :=, HighRange :=, LowRange :=, Tol :=, ActValue =>, WireBreakStatus =>, LowAlarmStatus =>, HighAlarmStatus =>, LoTol =>, HighTol =>, "4To20mA" =>)
   END_RUNG
   // the same network as SCL:
   #Ai18();   // "FB:Analog_Scaling"
END_REGION

REGION Network 19: #Ai19--AI SPARE 07
   RUNG wire#powerrail
      #Ai19(AnalogInputIw :=, AlmHighLimit :=, AlmLowlimit :=, Correction :=, SimValue :=, SimBit :=, HighRange :=, LowRange :=, Tol :=, ActValue =>, WireBreakStatus =>, LowAlarmStatus =>, HighAlarmStatus =>, LoTol =>, HighTol =>, "4To20mA" =>)
   END_RUNG
   // the same network as SCL:
   #Ai19();   // "FB:Analog_Scaling"
END_REGION

REGION Network 20: #Ai20--AI SPARE 08
   RUNG wire#powerrail
      #Ai20(AnalogInputIw :=, AlmHighLimit :=, AlmLowlimit :=, Correction :=, SimValue :=, SimBit :=, HighRange :=, LowRange :=, Tol :=, ActValue =>, WireBreakStatus =>, LowAlarmStatus =>, HighAlarmStatus =>, LoTol =>, HighTol =>, "4To20mA" =>)
   END_RUNG
   // the same network as SCL:
   #Ai20();   // "FB:Analog_Scaling"
END_REGION

REGION Network 21: #Ai21--AI SPARE 09
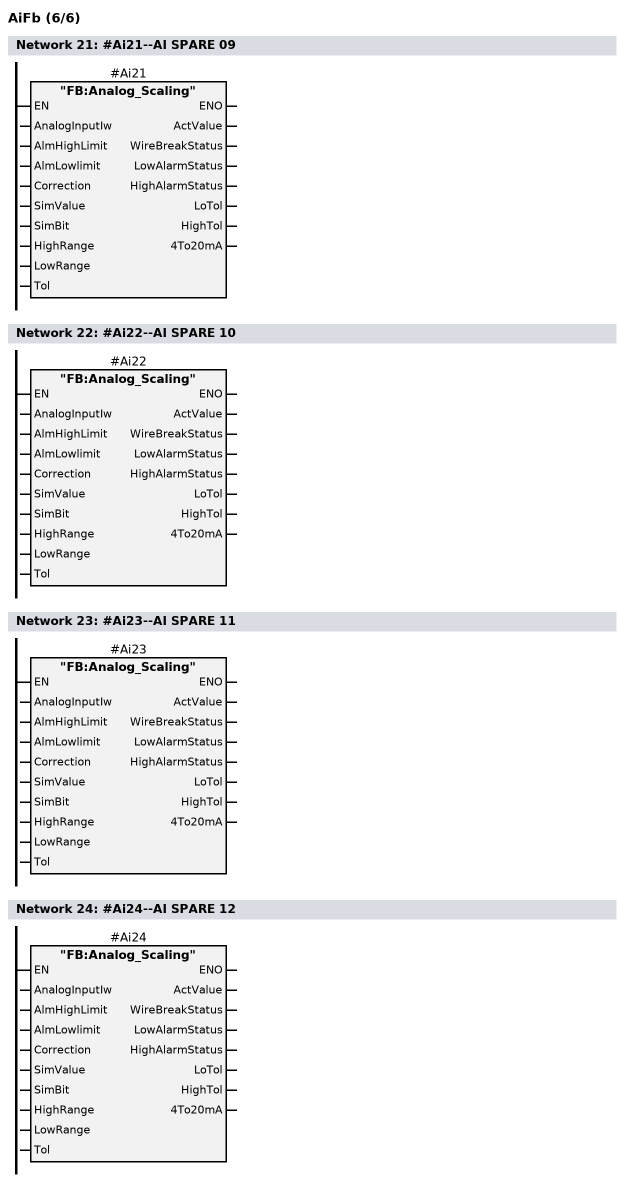
   RUNG wire#powerrail
      #Ai21(AnalogInputIw :=, AlmHighLimit :=, AlmLowlimit :=, Correction :=, SimValue :=, SimBit :=, HighRange :=, LowRange :=, Tol :=, ActValue =>, WireBreakStatus =>, LowAlarmStatus =>, HighAlarmStatus =>, LoTol =>, HighTol =>, "4To20mA" =>)
   END_RUNG
   // the same network as SCL:
   #Ai21();   // "FB:Analog_Scaling"
END_REGION

REGION Network 22: #Ai22--AI SPARE 10
   RUNG wire#powerrail
      #Ai22(AnalogInputIw :=, AlmHighLimit :=, AlmLowlimit :=, Correction :=, SimValue :=, SimBit :=, HighRange :=, LowRange :=, Tol :=, ActValue =>, WireBreakStatus =>, LowAlarmStatus =>, HighAlarmStatus =>, LoTol =>, HighTol =>, "4To20mA" =>)
   END_RUNG
   // the same network as SCL:
   #Ai22();   // "FB:Analog_Scaling"
END_REGION

REGION Network 23: #Ai23--AI SPARE 11
   RUNG wire#powerrail
      #Ai23(AnalogInputIw :=, AlmHighLimit :=, AlmLowlimit :=, Correction :=, SimValue :=, SimBit :=, HighRange :=, LowRange :=, Tol :=, ActValue =>, WireBreakStatus =>, LowAlarmStatus =>, HighAlarmStatus =>, LoTol =>, HighTol =>, "4To20mA" =>)
   END_RUNG
   // the same network as SCL:
   #Ai23();   // "FB:Analog_Scaling"
END_REGION

REGION Network 24: #Ai24--AI SPARE 12
   RUNG wire#powerrail
      #Ai24(AnalogInputIw :=, AlmHighLimit :=, AlmLowlimit :=, Correction :=, SimValue :=, SimBit :=, HighRange :=, LowRange :=, Tol :=, ActValue =>, WireBreakStatus =>, LowAlarmStatus =>, HighAlarmStatus =>, LoTol =>, HighTol =>, "4To20mA" =>)
   END_RUNG
   // the same network as SCL:
   #Ai24();   // "FB:Analog_Scaling"
END_REGION
END_FUNCTION_BLOCK

FUNCTION "AoFc" : Void   // FC106, LAD
{ S7_Optimized_Access := 'TRUE' }
// stored: AutoNumber false, SetENOAutomatically false
   VAR_TEMP   // added for the SCL form of the ladder/FBD networks
      _w1 : Bool;
      _w2 : Bool;
   END_VAR
BEGIN

REGION Network 1: "AoDb"
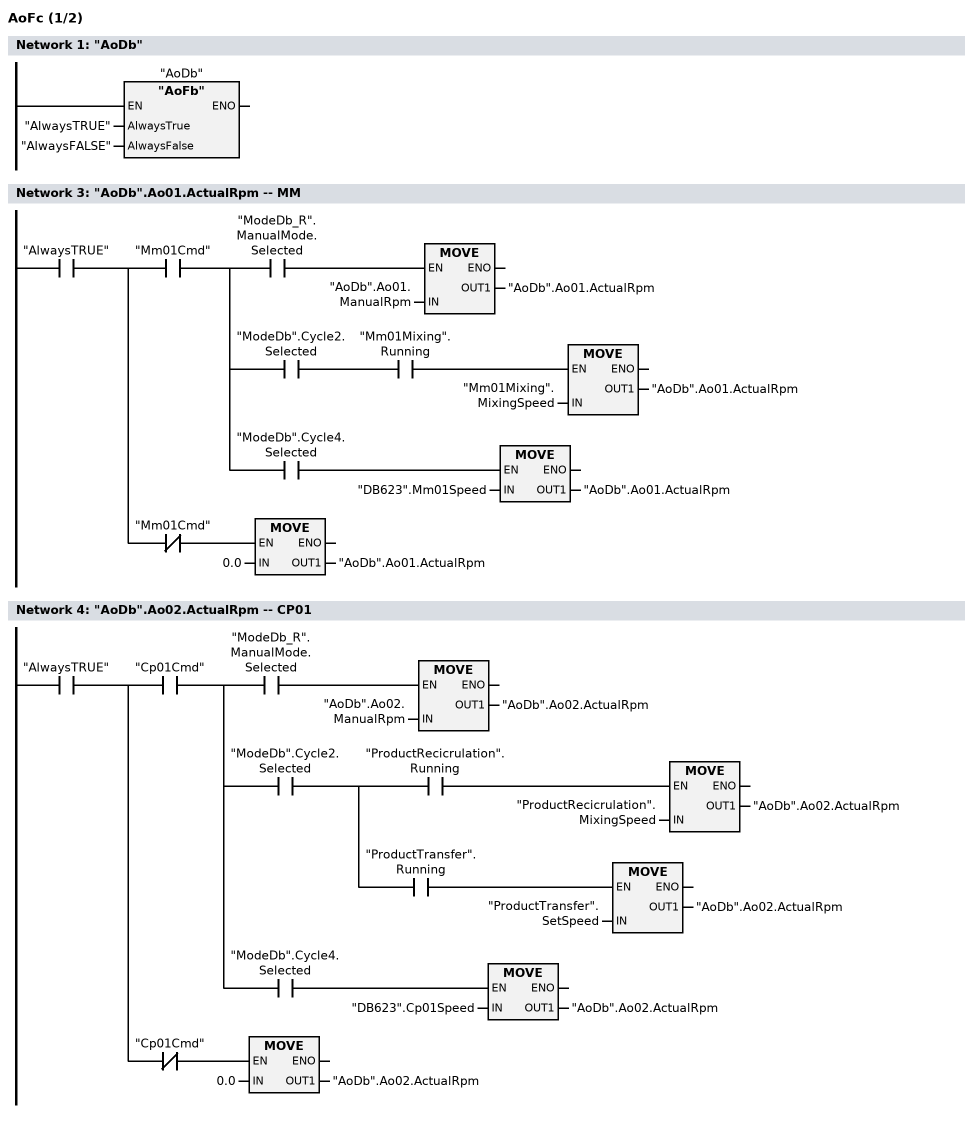
   RUNG wire#powerrail
      "AoDb"(AlwaysTrue := "AlwaysTRUE", AlwaysFalse := "AlwaysFALSE")
   END_RUNG
   // the same network as SCL:
   "AoDb"(AlwaysTrue := "AlwaysTRUE", AlwaysFalse := "AlwaysFALSE");   // "AoFb"
END_REGION

REGION Network 2 (SCL): Output to PLC Tag
   "Mm01Ref" := "AoDb".Ao01.Output;
   "Cp01Ref" := "AoDb".Ao02.Output;
   "Cv01"    :=  "AoDb".Ao03.Output;
   "AoSpare1" := "AoDb".Ao04.Output;
   "AoSpare2" := "AoDb".Ao05.Output;
   "AoSpare3" := "AoDb".Ao06.Output;
   "AoSpare4" := "AoDb".Ao07.Output;
   "AoSpare5" := "AoDb".Ao08.Output;
END_REGION

REGION Network 3: "AoDb".Ao01.ActualRpm -- MM
   RUNG wire#powerrail
      Contact( "AlwaysTRUE" )
      wire#w1
      Contact( "Mm01Cmd" )
      wire#w2
      Contact( "ModeDb_R".ManualMode.Selected )
      Move(in := "AoDb".Ao01.ManualRpm, out1 => "AoDb".Ao01.ActualRpm)
   END_RUNG
   RUNG wire#w2
      Contact( "ModeDb".Cycle2.Selected )
      Contact( "Mm01Mixing".Running )
      Move(in := "Mm01Mixing".MixingSpeed, out1 => "AoDb".Ao01.ActualRpm)
   END_RUNG
   RUNG wire#w2
      Contact( "ModeDb".Cycle4.Selected )
      Move(in := "DB623".Mm01Speed, out1 => "AoDb".Ao01.ActualRpm)
   END_RUNG
   RUNG wire#w1
      I_Contact( "Mm01Cmd" )
      Move(in := 0.0, out1 => "AoDb".Ao01.ActualRpm)
   END_RUNG
   // the same network as SCL:
   #_w1 := "AlwaysTRUE" AND "Mm01Cmd";
   IF #_w1 AND "ModeDb_R".ManualMode.Selected THEN "AoDb".Ao01.ActualRpm := "AoDb".Ao01.ManualRpm; END_IF;
   IF #_w1 AND "ModeDb".Cycle2.Selected AND "Mm01Mixing".Running THEN
       "AoDb".Ao01.ActualRpm := "Mm01Mixing".MixingSpeed;
   END_IF;
   IF #_w1 AND "ModeDb".Cycle4.Selected THEN "AoDb".Ao01.ActualRpm := "DB623".Mm01Speed; END_IF;
   IF "AlwaysTRUE" AND NOT "Mm01Cmd" THEN "AoDb".Ao01.ActualRpm := 0.0; END_IF;
END_REGION

REGION Network 4: "AoDb".Ao02.ActualRpm -- CP01
   RUNG wire#powerrail
      Contact( "AlwaysTRUE" )
      wire#w1
      Contact( "Cp01Cmd" )
      wire#w2
      Contact( "ModeDb_R".ManualMode.Selected )
      Move(in := "AoDb".Ao02.ManualRpm, out1 => "AoDb".Ao02.ActualRpm)
   END_RUNG
   RUNG wire#w2
      Contact( "ModeDb".Cycle2.Selected )
      wire#w3
      Contact( "ProductRecicrulation".Running )
      Move(in := "ProductRecicrulation".MixingSpeed, out1 => "AoDb".Ao02.ActualRpm)
   END_RUNG
   RUNG wire#w3
      Contact( "ProductTransfer".Running )
      Move(in := "ProductTransfer".SetSpeed, out1 => "AoDb".Ao02.ActualRpm)
   END_RUNG
   RUNG wire#w2
      Contact( "ModeDb".Cycle4.Selected )
      Move(in := "DB623".Cp01Speed, out1 => "AoDb".Ao02.ActualRpm)
   END_RUNG
   RUNG wire#w1
      I_Contact( "Cp01Cmd" )
      Move(in := 0.0, out1 => "AoDb".Ao02.ActualRpm)
   END_RUNG
   // the same network as SCL:
   #_w1 := "AlwaysTRUE" AND "Cp01Cmd";
   IF #_w1 AND "ModeDb_R".ManualMode.Selected THEN "AoDb".Ao02.ActualRpm := "AoDb".Ao02.ManualRpm; END_IF;
   #_w2 := #_w1 AND "ModeDb".Cycle2.Selected;
   IF #_w2 AND "ProductRecicrulation".Running THEN
       "AoDb".Ao02.ActualRpm := "ProductRecicrulation".MixingSpeed;
   END_IF;
   IF #_w2 AND "ProductTransfer".Running THEN "AoDb".Ao02.ActualRpm := "ProductTransfer".SetSpeed; END_IF;
   IF #_w1 AND "ModeDb".Cycle4.Selected THEN "AoDb".Ao02.ActualRpm := "DB623".Cp01Speed; END_IF;
   IF "AlwaysTRUE" AND NOT "Cp01Cmd" THEN "AoDb".Ao02.ActualRpm := 0.0; END_IF;
END_REGION

REGION Network 5: CV01
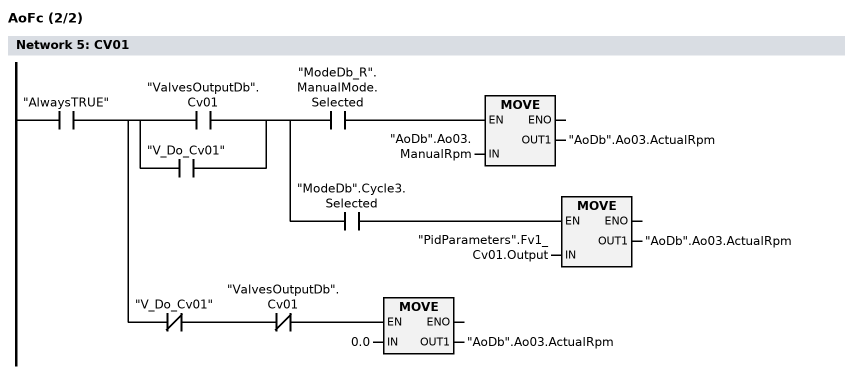
   RUNG wire#powerrail
      Contact( "AlwaysTRUE" )
      wire#w1
      Contact( "ValvesOutputDb".Cv01 )
      wire#w2
      Contact( "ModeDb_R".ManualMode.Selected )
      Move(in := "AoDb".Ao03.ManualRpm, out1 => "AoDb".Ao03.ActualRpm)
   END_RUNG
   RUNG wire#w1
      Contact( "V_Do_Cv01" )
   END_RUNG wire#w2
   RUNG wire#w2
      Contact( "ModeDb".Cycle3.Selected )
      Move(in := "PidParameters".Fv1_Cv01.Output, out1 => "AoDb".Ao03.ActualRpm)
   END_RUNG
   RUNG wire#w1
      I_Contact( "V_Do_Cv01" )
      I_Contact( "ValvesOutputDb".Cv01 )
      Move(in := 0.0, out1 => "AoDb".Ao03.ActualRpm)
   END_RUNG
   // the same network as SCL:
   #_w1 := "AlwaysTRUE" AND ("ValvesOutputDb".Cv01 OR "V_Do_Cv01");
   IF #_w1 AND "ModeDb_R".ManualMode.Selected THEN "AoDb".Ao03.ActualRpm := "AoDb".Ao03.ManualRpm; END_IF;
   IF #_w1 AND "ModeDb".Cycle3.Selected THEN
       "AoDb".Ao03.ActualRpm := "PidParameters".Fv1_Cv01.Output;
   END_IF;
   IF "AlwaysTRUE" AND NOT "V_Do_Cv01" AND NOT "ValvesOutputDb".Cv01 THEN
       "AoDb".Ao03.ActualRpm := 0.0;
   END_IF;
END_REGION
END_FUNCTION

FUNCTION_BLOCK "AoFb"   // FB106, LAD
{ S7_Optimized_Access := 'TRUE' }
// stored: AutoNumber false, MemoryReserve 100, SetENOAutomatically false
   VAR_INPUT
      AlwaysTrue : Bool;
      AlwaysFalse : Bool;
   END_VAR
   VAR
      Ao01 { S7_SetPoint := 'True'} : "AnalogOutputScaling";   // Mm01Ref
      Ao02 { S7_SetPoint := 'True'} : "AnalogOutputScaling";   // Cp01Ref
      Ao03 { S7_SetPoint := 'True'} : "AnalogOutputScaling";   // Cv01
      Ao04 { S7_SetPoint := 'True'} : "AnalogOutputScaling";   // AoSpare1
      Ao05 { S7_SetPoint := 'True'} : "AnalogOutputScaling";   // AoSpare2
      Ao06 { S7_SetPoint := 'True'} : "AnalogOutputScaling";   // AoSpare3
      Ao07 { S7_SetPoint := 'True'} : "AnalogOutputScaling";   // AoSpare4
      Ao08 { S7_SetPoint := 'True'} : "AnalogOutputScaling";   // AoSpare5
   END_VAR
BEGIN

REGION Network 2: Mm01Ref
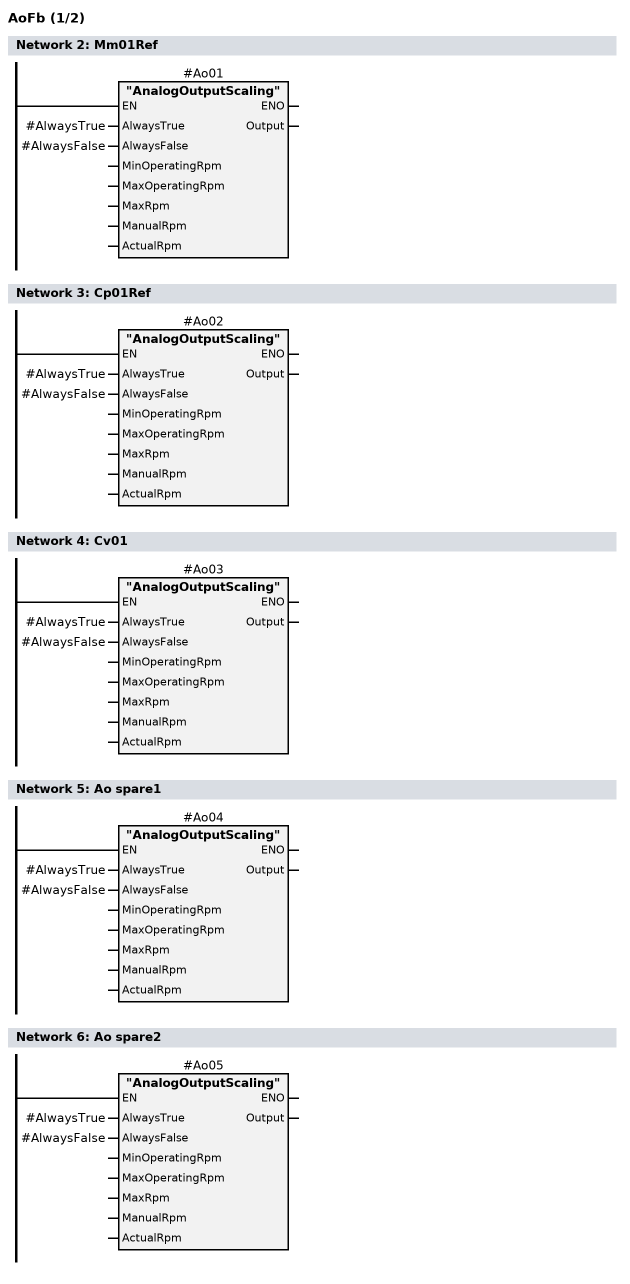
   RUNG wire#powerrail
      #Ao01(AlwaysTrue := #AlwaysTrue, AlwaysFalse := #AlwaysFalse, MinOperatingRpm :=, MaxOperatingRpm :=, MaxRpm :=, ManualRpm :=, ActualRpm :=, Output =>)
   END_RUNG
   // the same network as SCL:
   #Ao01(AlwaysTrue := #AlwaysTrue, AlwaysFalse := #AlwaysFalse);   // "AnalogOutputScaling"
END_REGION

REGION Network 3: Cp01Ref
   RUNG wire#powerrail
      #Ao02(AlwaysTrue := #AlwaysTrue, AlwaysFalse := #AlwaysFalse, MinOperatingRpm :=, MaxOperatingRpm :=, MaxRpm :=, ManualRpm :=, ActualRpm :=, Output =>)
   END_RUNG
   // the same network as SCL:
   #Ao02(AlwaysTrue := #AlwaysTrue, AlwaysFalse := #AlwaysFalse);   // "AnalogOutputScaling"
END_REGION

REGION Network 4: Cv01
   RUNG wire#powerrail
      #Ao03(AlwaysTrue := #AlwaysTrue, AlwaysFalse := #AlwaysFalse, MinOperatingRpm :=, MaxOperatingRpm :=, MaxRpm :=, ManualRpm :=, ActualRpm :=, Output =>)
   END_RUNG
   // the same network as SCL:
   #Ao03(AlwaysTrue := #AlwaysTrue, AlwaysFalse := #AlwaysFalse);   // "AnalogOutputScaling"
END_REGION

REGION Network 5: Ao spare1
   RUNG wire#powerrail
      #Ao04(AlwaysTrue := #AlwaysTrue, AlwaysFalse := #AlwaysFalse, MinOperatingRpm :=, MaxOperatingRpm :=, MaxRpm :=, ManualRpm :=, ActualRpm :=, Output =>)
   END_RUNG
   // the same network as SCL:
   #Ao04(AlwaysTrue := #AlwaysTrue, AlwaysFalse := #AlwaysFalse);   // "AnalogOutputScaling"
END_REGION

REGION Network 6: Ao spare2
   RUNG wire#powerrail
      #Ao05(AlwaysTrue := #AlwaysTrue, AlwaysFalse := #AlwaysFalse, MinOperatingRpm :=, MaxOperatingRpm :=, MaxRpm :=, ManualRpm :=, ActualRpm :=, Output =>)
   END_RUNG
   // the same network as SCL:
   #Ao05(AlwaysTrue := #AlwaysTrue, AlwaysFalse := #AlwaysFalse);   // "AnalogOutputScaling"
END_REGION

REGION Network 7: Ao spare3
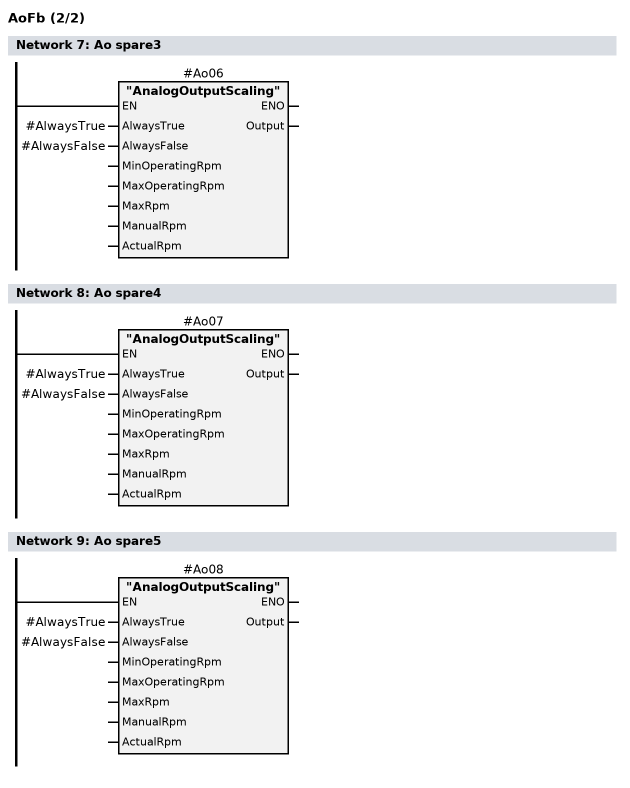
   RUNG wire#powerrail
      #Ao06(AlwaysTrue := #AlwaysTrue, AlwaysFalse := #AlwaysFalse, MinOperatingRpm :=, MaxOperatingRpm :=, MaxRpm :=, ManualRpm :=, ActualRpm :=, Output =>)
   END_RUNG
   // the same network as SCL:
   #Ao06(AlwaysTrue := #AlwaysTrue, AlwaysFalse := #AlwaysFalse);   // "AnalogOutputScaling"
END_REGION

REGION Network 8: Ao spare4
   RUNG wire#powerrail
      #Ao07(AlwaysTrue := #AlwaysTrue, AlwaysFalse := #AlwaysFalse, MinOperatingRpm :=, MaxOperatingRpm :=, MaxRpm :=, ManualRpm :=, ActualRpm :=, Output =>)
   END_RUNG
   // the same network as SCL:
   #Ao07(AlwaysTrue := #AlwaysTrue, AlwaysFalse := #AlwaysFalse);   // "AnalogOutputScaling"
END_REGION

REGION Network 9: Ao spare5
   RUNG wire#powerrail
      #Ao08(AlwaysTrue := #AlwaysTrue, AlwaysFalse := #AlwaysFalse, MinOperatingRpm :=, MaxOperatingRpm :=, MaxRpm :=, ManualRpm :=, ActualRpm :=, Output =>)
   END_RUNG
   // the same network as SCL:
   #Ao08(AlwaysTrue := #AlwaysTrue, AlwaysFalse := #AlwaysFalse);   // "AnalogOutputScaling"
END_REGION
END_FUNCTION_BLOCK

FUNCTION_BLOCK "AnalogOutputScaling"   // FB11, LAD
{ S7_Optimized_Access := 'FALSE' }
// stored: SetENOAutomatically false
   VAR_INPUT
      AlwaysTrue : Bool;
      AlwaysFalse : Bool;
      MinOperatingRpm : Real;
      MaxOperatingRpm : Real;
      MaxRpm : Real;
      ManualRpm : Real;
      ActualRpm : Real;
   END_VAR
   VAR_OUTPUT
      Output : Int;
   END_VAR
   VAR
      Temp : Real;
   END_VAR
BEGIN

REGION Network 1: Scaling
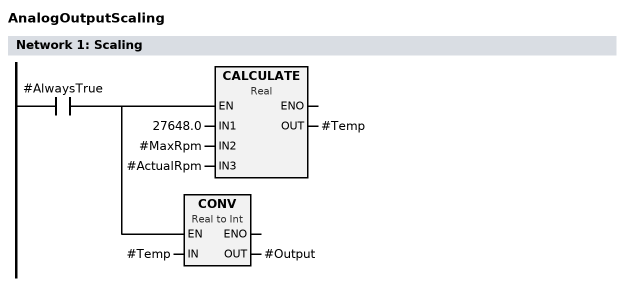
   RUNG wire#powerrail
      Contact( #AlwaysTrue )
      wire#w1
      { S7_Templates := "SrcType := Real"; S7_GenerateENO := "TRUE"; S7_Expression := "(in1*IN3)/IN2" } Calculate(in1 := 27648.0, in2 := #MaxRpm, in3 := #ActualRpm, out => #Temp)
   END_RUNG
   RUNG wire#w1
      { S7_Templates := "[SrcType := Real, DestType := Int]"; S7_GenerateENO := "TRUE" } Convert(in := #Temp, out => #Output)
   END_RUNG
   // the same network as SCL:
   IF #AlwaysTrue THEN
       #Temp := (27648.0*#ActualRpm)/#MaxRpm;
       #Output := REAL_TO_INT(#Temp);
   END_IF;
END_REGION
END_FUNCTION_BLOCK

FUNCTION "DiFc" : Void   // FC101, LAD
TITLE = DIFC
{ S7_Optimized_Access := 'TRUE' }
// stored: AutoNumber false, SetENOAutomatically false
BEGIN

REGION Network 1 (SCL): DI Final
   "DiFinal".ControlKey := "DiSimulation".ControlKey OR "ControlKey";
   "DiFinal".EmergencyStop := "DiSimulation".EmergencyStop OR "EmergencyStop";
   "DiFinal".CompressedAirPressureLow := "DiSimulation".CompressedAirPressureLow OR "CompressedAirPressureLow";
   "DiFinal".PowerFailure := "DiSimulation".PowerFailure OR "PowerFailure";
   "DiFinal".PowerReset := "DiSimulation".PowerReset OR "PowerReset";
   "DiFinal".MagneticMixerFeedback := "DiSimulation".MagneticMixerFeedback OR "MagneticMixerFeedback";
   "DiFinal".CipPumpFeedback := "DiSimulation".CipPumpFeedback OR "CipPumpFeedback";
   "DiFinal".MagneticMixerOverload := "DiSimulation".MagneticMixerOverload OR "MagneticMixerOverload";
   "DiFinal".CipPumpOverload := "DiSimulation".CipPumpOverload OR "CipPumpOverload";
   "DiFinal".RuptureDisc := "DiSimulation".RuptureDisc OR "RuptureDisc";
   "DiFinal".Cp01FlowSwitch := "DiSimulation".Cp01FlowSwitch OR "Cp01FlowSwitch";
   "DiFinal".DiSpare1 := "DiSimulation".DiSpare1 OR "DiSpare1";
   "DiFinal".DiSpare2 := "DiSimulation".DiSpare2 OR "DiSpare2";
   "DiFinal".MMHighSpeedSensor := "DiSimulation".MMHighSpeedSensor OR "MMHighSpeedSensor";
   "DiFinal".DiSpare3 := "DiSimulation".DiSpare3 OR "DiSpare3";
   "DiFinal".DiSpare4 := "DiSimulation".DiSpare4 OR "DiSpare4";
   "DiFinal".DiSpare5 := "DiSimulation".DiSpare5 OR "DiSpare5";
   "DiFinal".DiSpare6 := "DiSimulation".DiSpare6 OR "DiSpare6";
   "DiFinal".DiSpare7 := "DiSimulation".DiSpare7 OR "DiSpare7";
   "DiFinal".DiSpare8 := "DiSimulation".DiSpare8 OR "DiSpare8";
   "DiFinal".DiSpare9:= "DiSimulation".DiSpare9 OR "DiSpare9";
   "DiFinal".DiSpare10 := "DiSimulation".DiSpare10 OR "DiSpare10";
END_REGION
END_FUNCTION

FUNCTION "DoFc" : Void   // FC109, LAD
{ S7_Optimized_Access := 'FALSE' }
// stored: AutoNumber false, SetENOAutomatically false
   VAR_TEMP   // added for the SCL form of the ladder/FBD networks
      _w1 : Bool;
   END_VAR
BEGIN

REGION Network 2: "DoDb"
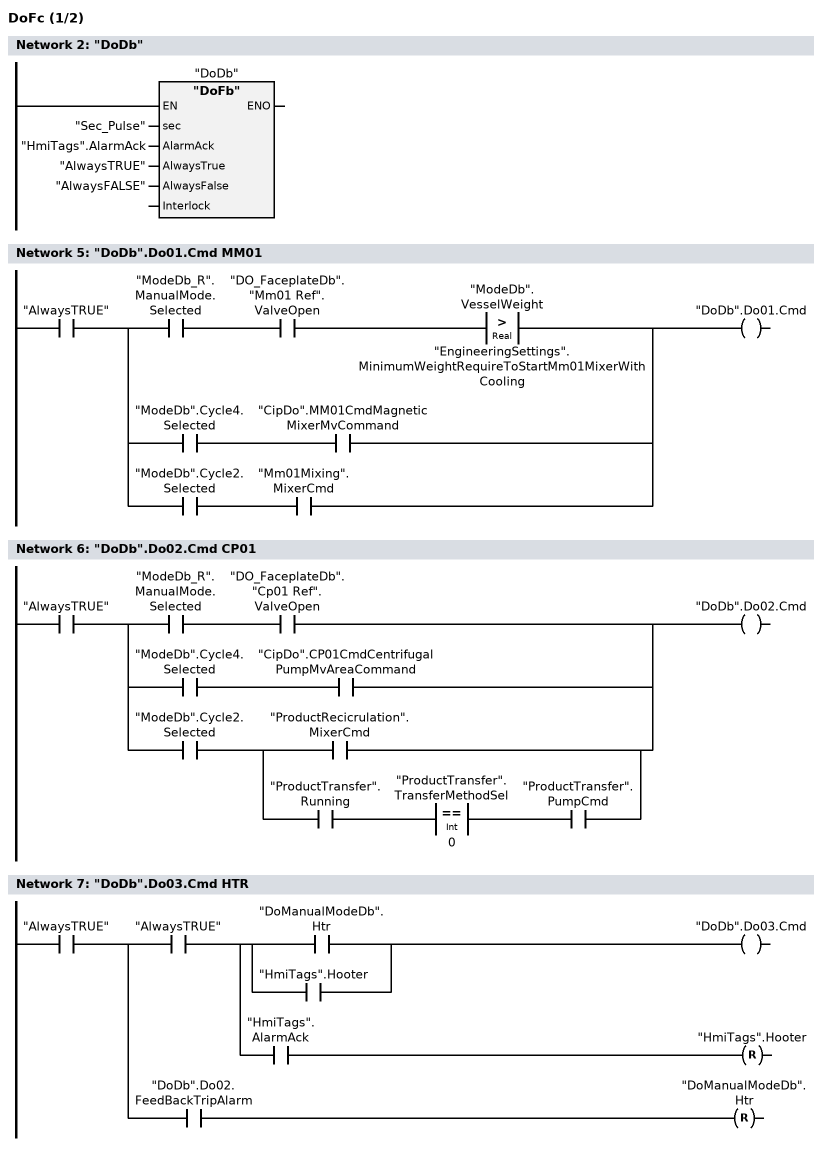
   RUNG wire#powerrail
      "DoDb"(sec := "Sec_Pulse", AlarmAck := "HmiTags".AlarmAck, AlwaysTrue := "AlwaysTRUE", AlwaysFalse := "AlwaysFALSE", Interlock :=)
   END_RUNG
   // the same network as SCL:
   "DoDb"(sec := "Sec_Pulse",   // "DoFb"
          AlarmAck := "HmiTags".AlarmAck,
          AlwaysTrue := "AlwaysTRUE",
          AlwaysFalse := "AlwaysFALSE");
END_REGION

REGION Network 3 (SCL): Digital Output
   "Mm01Cmd":= "DoDb".Do01."Output";
   "Cp01Cmd" := "DoDb".Do02."Output";
   "Htr" := "DoDb".Do03."Output" OR "DoDb".Do03.Cmd;
   "Lf01" := "DoDb".Do04."Output" OR "DoDb".Do04.Cmd;
   "DoSpare1" := "DoDb".Do05."Output";
   "DoSpare2" := "DoDb".Do06."Output";
   "DoSpare3" := "DoDb".Do07."Output";
   "DoSpare4" := "DoDb".Do08."Output";
   "DoSpare5" := "DoDb".Do09."Output";
   "DoSpare6" := "DoDb".Do10."Output";
END_REGION

REGION Network 4 (SCL): MANUAL MODE SELECTED
   //"DoDb".Do01.ManualModeSelected := "ModeDb".MV5000.Mode.ManualMode.Selected;
   "DoDb".Do01.ModeSel := "ModeDb_R".ManualMode.Selected;
   "DoDb".Do02.ModeSel := "ModeDb_R".ManualMode.Selected;
   "DoDb".Do03.ModeSel := "ModeDb_R".ManualMode.Selected;
   "DoDb".Do04.ModeSel := "ModeDb_R".ManualMode.Selected;
   "DoDb".Do05.ModeSel := "ModeDb_R".ManualMode.Selected;
END_REGION

REGION Network 5: "DoDb".Do01.Cmd MM01
   RUNG wire#powerrail
      Contact( "AlwaysTRUE" )
      wire#w1
      Contact( "ModeDb_R".ManualMode.Selected )
      Contact( "DO_FaceplateDb"."Mm01 Ref".ValveOpen )
      { S7_Templates := "SrcType := Real" } GT_Contact(in1 := "ModeDb".VesselWeight, in2 := "EngineeringSettings".MinimumWeightRequireToStartMm01MixerWithCooling)
      wire#w2
      Coil( "DoDb".Do01.Cmd )
   END_RUNG
   RUNG wire#w1
      Contact( "ModeDb".Cycle4.Selected )
      Contact( "CipDo".MM01CmdMagneticMixerMvCommand )
   END_RUNG wire#w2
   RUNG wire#w1
      Contact( "ModeDb".Cycle2.Selected )
      Contact( "Mm01Mixing".MixerCmd )
   END_RUNG wire#w2
   // the same network as SCL:
   "DoDb".Do01.Cmd := "AlwaysTRUE" AND (("ModeDb_R".ManualMode.Selected AND "DO_FaceplateDb"."Mm01 Ref".ValveOpen AND ("ModeDb".VesselWeight > "EngineeringSettings".MinimumWeightRequireToStartMm01MixerWithCooling)) OR ("ModeDb".Cycle4.Selected AND "CipDo".MM01CmdMagneticMixerMvCommand) OR ("ModeDb".Cycle2.Selected AND "Mm01Mixing".MixerCmd));
END_REGION

REGION Network 6: "DoDb".Do02.Cmd CP01
   RUNG wire#powerrail
      Contact( "AlwaysTRUE" )
      wire#w1
      Contact( "ModeDb_R".ManualMode.Selected )
      Contact( "DO_FaceplateDb"."Cp01 Ref".ValveOpen )
      wire#w2
      Coil( "DoDb".Do02.Cmd )
   END_RUNG
   RUNG wire#w1
      Contact( "ModeDb".Cycle4.Selected )
      Contact( "CipDo".CP01CmdCentrifugalPumpMvAreaCommand )
   END_RUNG wire#w2
   RUNG wire#w1
      Contact( "ModeDb".Cycle2.Selected )
      wire#w3
      Contact( "ProductRecicrulation".MixerCmd )
   END_RUNG wire#w2
   RUNG wire#w3
      Contact( "ProductTransfer".Running )
      { S7_Templates := "SrcType := Int" } EQ_Contact(in1 := "ProductTransfer".TransferMethodSel, in2 := 0)
      Contact( "ProductTransfer".PumpCmd )
   END_RUNG wire#w2
   // the same network as SCL:
   "DoDb".Do02.Cmd := "AlwaysTRUE" AND (("ModeDb_R".ManualMode.Selected AND "DO_FaceplateDb"."Cp01 Ref".ValveOpen) OR ("ModeDb".Cycle4.Selected AND "CipDo".CP01CmdCentrifugalPumpMvAreaCommand) OR ("ModeDb".Cycle2.Selected AND ("ProductRecicrulation".MixerCmd OR ("ProductTransfer".Running AND ("ProductTransfer".TransferMethodSel = 0) AND "ProductTransfer".PumpCmd))));
END_REGION

REGION Network 7: "DoDb".Do03.Cmd HTR
   RUNG wire#powerrail
      Contact( "AlwaysTRUE" )
      wire#w1
      Contact( "AlwaysTRUE" )
      wire#w2
      Contact( "DoManualModeDb".Htr )
      wire#w3
      Coil( "DoDb".Do03.Cmd )
   END_RUNG
   RUNG wire#w2
      Contact( "HmiTags".Hooter )
   END_RUNG wire#w3
   RUNG wire#w2
      Contact( "HmiTags".AlarmAck )
      R_Coil( "HmiTags".Hooter )
   END_RUNG
   RUNG wire#w1
      Contact( "DoDb".Do02.FeedBackTripAlarm )
      R_Coil( "DoManualModeDb".Htr )
   END_RUNG
   // the same network as SCL:
   #_w1 := "AlwaysTRUE" AND "AlwaysTRUE";
   "DoDb".Do03.Cmd := #_w1 AND ("DoManualModeDb".Htr OR "HmiTags".Hooter);
   IF #_w1 AND "HmiTags".AlarmAck THEN "HmiTags".Hooter := FALSE; END_IF;
   IF "AlwaysTRUE" AND "DoDb".Do02.FeedBackTripAlarm THEN "DoManualModeDb".Htr := FALSE; END_IF;
END_REGION

REGION Network 8: "DoDb".Do04.Cmd
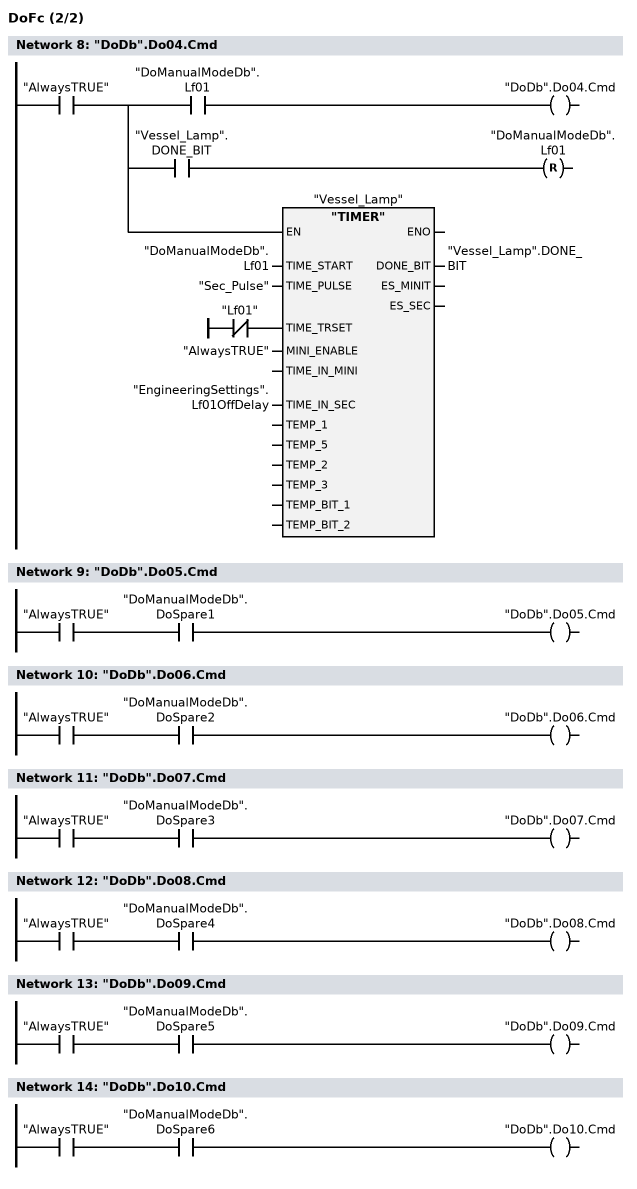
   RUNG wire#powerrail
      Contact( "AlwaysTRUE" )
      wire#w1
      Contact( "DoManualModeDb".Lf01 )
      Coil( "DoDb".Do04.Cmd )
   END_RUNG
   RUNG wire#w1
      Contact( "Vessel_Lamp".DONE_BIT )
      R_Coil( "DoManualModeDb".Lf01 )
   END_RUNG
   RUNG wire#w1
      "Vessel_Lamp"(TIME_TRSET := wire#w2, TIME_START := "DoManualModeDb".Lf01, TIME_PULSE := "Sec_Pulse", MINI_ENABLE := "AlwaysTRUE", TIME_IN_MINI :=, TIME_IN_SEC := "EngineeringSettings".Lf01OffDelay, TEMP_1 :=, TEMP_5 :=, TEMP_2 :=, TEMP_3 :=, TEMP_BIT_1 :=, TEMP_BIT_2 :=, DONE_BIT => "Vessel_Lamp".DONE_BIT, ES_MINIT =>, ES_SEC =>)
   END_RUNG
   RUNG wire#powerrail
      I_Contact( "Lf01" )
   END_RUNG wire#w2
   // the same network as SCL:
   "DoDb".Do04.Cmd := "AlwaysTRUE" AND "DoManualModeDb".Lf01;
   IF "AlwaysTRUE" AND "Vessel_Lamp".DONE_BIT THEN "DoManualModeDb".Lf01 := FALSE; END_IF;
   IF "AlwaysTRUE" THEN
       "Vessel_Lamp"(TIME_START := "DoManualModeDb".Lf01,   // "TIMER"
                     TIME_PULSE := "Sec_Pulse",
                     TIME_TRSET := NOT "Lf01",
                     MINI_ENABLE := "AlwaysTRUE",
                     TIME_IN_SEC := "EngineeringSettings".Lf01OffDelay,
                     DONE_BIT => "Vessel_Lamp".DONE_BIT);
   END_IF;
END_REGION

REGION Network 9: "DoDb".Do05.Cmd
   RUNG wire#powerrail
      Contact( "AlwaysTRUE" )
      Contact( "DoManualModeDb".DoSpare1 )
      Coil( "DoDb".Do05.Cmd )
   END_RUNG
   // the same network as SCL:
   "DoDb".Do05.Cmd := "AlwaysTRUE" AND "DoManualModeDb".DoSpare1;
END_REGION

REGION Network 10: "DoDb".Do06.Cmd
   RUNG wire#powerrail
      Contact( "AlwaysTRUE" )
      Contact( "DoManualModeDb".DoSpare2 )
      Coil( "DoDb".Do06.Cmd )
   END_RUNG
   // the same network as SCL:
   "DoDb".Do06.Cmd := "AlwaysTRUE" AND "DoManualModeDb".DoSpare2;
END_REGION

REGION Network 11: "DoDb".Do07.Cmd
   RUNG wire#powerrail
      Contact( "AlwaysTRUE" )
      Contact( "DoManualModeDb".DoSpare3 )
      Coil( "DoDb".Do07.Cmd )
   END_RUNG
   // the same network as SCL:
   "DoDb".Do07.Cmd := "AlwaysTRUE" AND "DoManualModeDb".DoSpare3;
END_REGION

REGION Network 12: "DoDb".Do08.Cmd
   RUNG wire#powerrail
      Contact( "AlwaysTRUE" )
      Contact( "DoManualModeDb".DoSpare4 )
      Coil( "DoDb".Do08.Cmd )
   END_RUNG
   // the same network as SCL:
   "DoDb".Do08.Cmd := "AlwaysTRUE" AND "DoManualModeDb".DoSpare4;
END_REGION

REGION Network 13: "DoDb".Do09.Cmd
   RUNG wire#powerrail
      Contact( "AlwaysTRUE" )
      Contact( "DoManualModeDb".DoSpare5 )
      Coil( "DoDb".Do09.Cmd )
   END_RUNG
   // the same network as SCL:
   "DoDb".Do09.Cmd := "AlwaysTRUE" AND "DoManualModeDb".DoSpare5;
END_REGION

REGION Network 14: "DoDb".Do10.Cmd
   RUNG wire#powerrail
      Contact( "AlwaysTRUE" )
      Contact( "DoManualModeDb".DoSpare6 )
      Coil( "DoDb".Do10.Cmd )
   END_RUNG
   // the same network as SCL:
   "DoDb".Do10.Cmd := "AlwaysTRUE" AND "DoManualModeDb".DoSpare6;
END_REGION

REGION Network 15 (SCL): Fb delay
   "DoDb".Do01.FBCheckDelay := "EngineeringSettings"."Mm01F/BDelay";
   "DoDb".Do02.FBCheckDelay := "EngineeringSettings"."Cp01F/BDelay";
   //"VesselLamp_DB".LF01.TIME_IN_SEC := "EngineeringSettings".Lf01OffDelay;
END_REGION

REGION Network 16 (SCL): FeedBack Alarms And Input
   "DoDb".Do01.MotorFeedbackInputSelection := 1;
   "DoDb".Do02.MotorFeedbackInputSelection := 1;

   "DoDb".Do01.MotorFeedbackInput := "DiFinal".MagneticMixerFeedback;
   "DoDb".Do02.MotorFeedbackInput := "DiFinal".CipPumpFeedback;

   "DoDb".Do02.FeedBackTripAlarm := "SafetyAlarms".Cp01FeedbackTrip;
   "DoDb".Do01.FeedBackTripAlarm := "SafetyAlarms".Mm01FeedbackTrip;


   "SafetyAlarms".Mm01FeedbackTrip := "DoDb".Do01.FeedBackTripAlarm;
   "SafetyAlarms".Cp01FeedbackTrip := "DoDb".Do02.FeedBackTripAlarm;

   "SafetyAlarms".Mm01FeedbackTrip := "DoDb".Do01.OpFbTrip;
   "SafetyAlarms".Cp01FeedbackTrip := "DoDb".Do02.OpFbTrip;

   "DoDb".Do01.AlarmAck := "HmiTags".AlarmAck;
   "DoDb".Do02.AlarmAck := "HmiTags".AlarmAck;
END_REGION
END_FUNCTION

FUNCTION_BLOCK "DoFb"   // FB109, LAD
{ S7_Optimized_Access := 'FALSE' }
// stored: AutoNumber false, SetENOAutomatically false
   VAR_INPUT
      sec : Bool;
      AlarmAck : Bool;
      AlwaysTrue : Bool;
      AlwaysFalse : Bool;
      Interlock : Bool;
   END_VAR
   VAR
      Do01 { S7_SetPoint := 'True'} : "DigitalOutput";   // Mm01Cmd
      Do02 { S7_SetPoint := 'True'} : "DigitalOutput";   // Cp01Cmd
      Do03 { S7_SetPoint := 'True'} : "DigitalOutput";   // Htr
      Do04 { S7_SetPoint := 'True'} : "DigitalOutput";   // Lf01
      Do05 { S7_SetPoint := 'True'} : "DigitalOutput";   // DoSpare1
      Do06 { S7_SetPoint := 'True'} : "DigitalOutput";   // DoSpare2
      Do07 { S7_SetPoint := 'True'} : "DigitalOutput";   // DoSpare3
      Do08 { S7_SetPoint := 'True'} : "DigitalOutput";   // DoSpare4
      Do09 { S7_SetPoint := 'True'} : "DigitalOutput";   // DoSpare5
      Do10 { S7_SetPoint := 'True'} : "DigitalOutput";   // DoSpare6
   END_VAR
BEGIN

REGION Network 1: Mm01Cmd
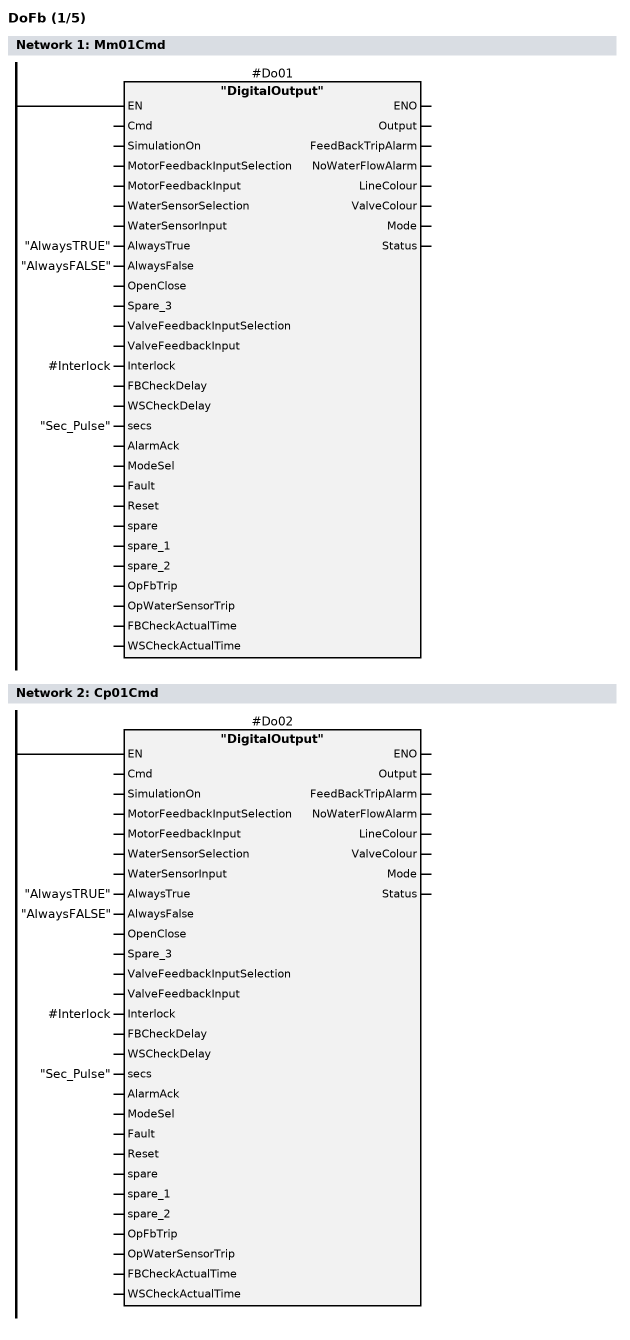
   RUNG wire#powerrail
      #Do01(Cmd :=, SimulationOn :=, MotorFeedbackInputSelection :=, MotorFeedbackInput :=, WaterSensorSelection :=, WaterSensorInput :=, AlwaysTrue := "AlwaysTRUE", AlwaysFalse := "AlwaysFALSE", OpenClose :=, Spare_3 :=, ValveFeedbackInputSelection :=, ValveFeedbackInput :=, Interlock := #Interlock, FBCheckDelay :=, WSCheckDelay :=, secs := "Sec_Pulse", AlarmAck :=, ModeSel :=, Fault :=, Reset :=, spare :=, spare_1 :=, spare_2 :=, OpFbTrip :=, OpWaterSensorTrip :=, FBCheckActualTime :=, WSCheckActualTime :=, Output =>, FeedBackTripAlarm =>, NoWaterFlowAlarm =>, LineColour =>, ValveColour =>, Mode =>, Status =>)
   END_RUNG
   // the same network as SCL:
   #Do01(AlwaysTrue := "AlwaysTRUE", AlwaysFalse := "AlwaysFALSE", Interlock := #Interlock, secs := "Sec_Pulse");   // "DigitalOutput"
END_REGION

REGION Network 2: Cp01Cmd
   RUNG wire#powerrail
      #Do02(Cmd :=, SimulationOn :=, MotorFeedbackInputSelection :=, MotorFeedbackInput :=, WaterSensorSelection :=, WaterSensorInput :=, AlwaysTrue := "AlwaysTRUE", AlwaysFalse := "AlwaysFALSE", OpenClose :=, Spare_3 :=, ValveFeedbackInputSelection :=, ValveFeedbackInput :=, Interlock := #Interlock, FBCheckDelay :=, WSCheckDelay :=, secs := "Sec_Pulse", AlarmAck :=, ModeSel :=, Fault :=, Reset :=, spare :=, spare_1 :=, spare_2 :=, OpFbTrip :=, OpWaterSensorTrip :=, FBCheckActualTime :=, WSCheckActualTime :=, Output =>, FeedBackTripAlarm =>, NoWaterFlowAlarm =>, LineColour =>, ValveColour =>, Mode =>, Status =>)
   END_RUNG
   // the same network as SCL:
   #Do02(AlwaysTrue := "AlwaysTRUE", AlwaysFalse := "AlwaysFALSE", Interlock := #Interlock, secs := "Sec_Pulse");   // "DigitalOutput"
END_REGION

REGION Network 3: Htr
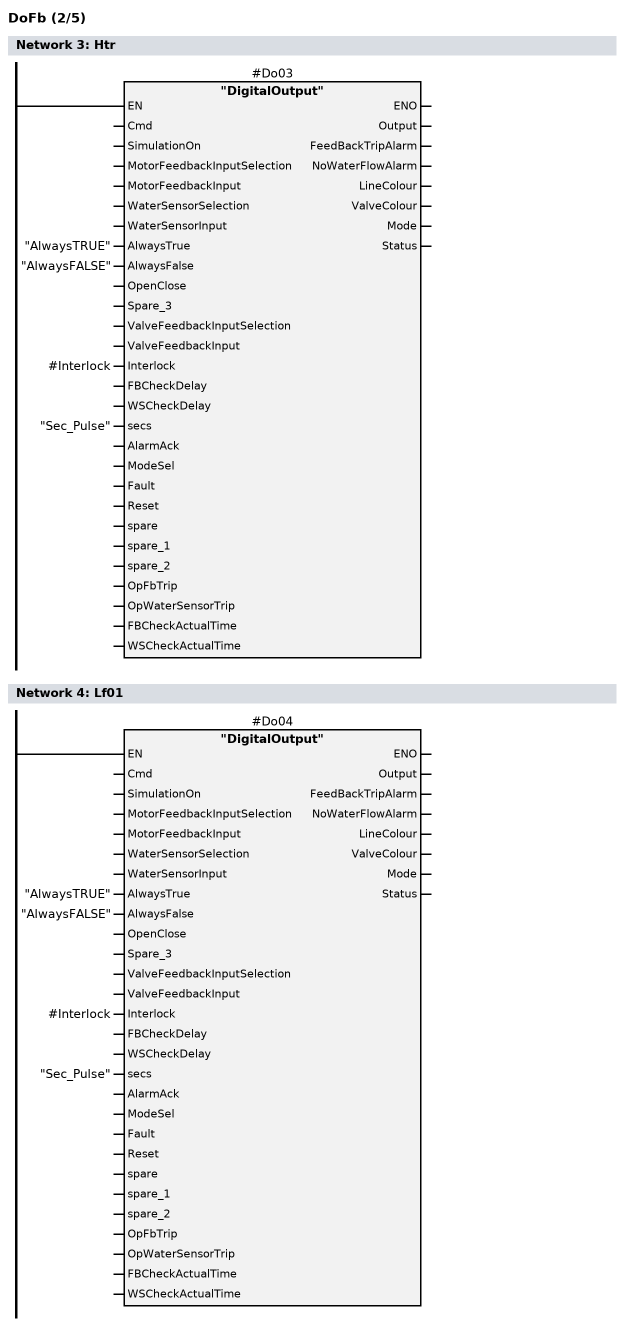
   RUNG wire#powerrail
      #Do03(Cmd :=, SimulationOn :=, MotorFeedbackInputSelection :=, MotorFeedbackInput :=, WaterSensorSelection :=, WaterSensorInput :=, AlwaysTrue := "AlwaysTRUE", AlwaysFalse := "AlwaysFALSE", OpenClose :=, Spare_3 :=, ValveFeedbackInputSelection :=, ValveFeedbackInput :=, Interlock := #Interlock, FBCheckDelay :=, WSCheckDelay :=, secs := "Sec_Pulse", AlarmAck :=, ModeSel :=, Fault :=, Reset :=, spare :=, spare_1 :=, spare_2 :=, OpFbTrip :=, OpWaterSensorTrip :=, FBCheckActualTime :=, WSCheckActualTime :=, Output =>, FeedBackTripAlarm =>, NoWaterFlowAlarm =>, LineColour =>, ValveColour =>, Mode =>, Status =>)
   END_RUNG
   // the same network as SCL:
   #Do03(AlwaysTrue := "AlwaysTRUE", AlwaysFalse := "AlwaysFALSE", Interlock := #Interlock, secs := "Sec_Pulse");   // "DigitalOutput"
END_REGION

REGION Network 4: Lf01
   RUNG wire#powerrail
      #Do04(Cmd :=, SimulationOn :=, MotorFeedbackInputSelection :=, MotorFeedbackInput :=, WaterSensorSelection :=, WaterSensorInput :=, AlwaysTrue := "AlwaysTRUE", AlwaysFalse := "AlwaysFALSE", OpenClose :=, Spare_3 :=, ValveFeedbackInputSelection :=, ValveFeedbackInput :=, Interlock := #Interlock, FBCheckDelay :=, WSCheckDelay :=, secs := "Sec_Pulse", AlarmAck :=, ModeSel :=, Fault :=, Reset :=, spare :=, spare_1 :=, spare_2 :=, OpFbTrip :=, OpWaterSensorTrip :=, FBCheckActualTime :=, WSCheckActualTime :=, Output =>, FeedBackTripAlarm =>, NoWaterFlowAlarm =>, LineColour =>, ValveColour =>, Mode =>, Status =>)
   END_RUNG
   // the same network as SCL:
   #Do04(AlwaysTrue := "AlwaysTRUE", AlwaysFalse := "AlwaysFALSE", Interlock := #Interlock, secs := "Sec_Pulse");   // "DigitalOutput"
END_REGION

REGION Network 5: #Do05 spare1
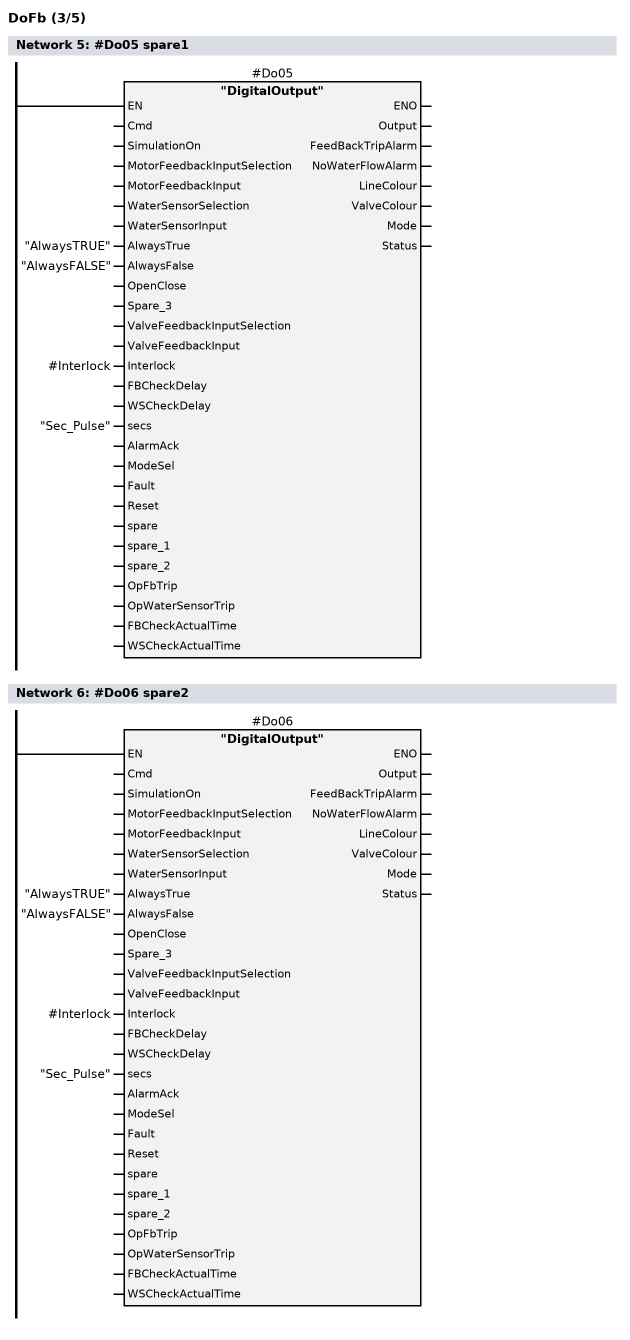
   RUNG wire#powerrail
      #Do05(Cmd :=, SimulationOn :=, MotorFeedbackInputSelection :=, MotorFeedbackInput :=, WaterSensorSelection :=, WaterSensorInput :=, AlwaysTrue := "AlwaysTRUE", AlwaysFalse := "AlwaysFALSE", OpenClose :=, Spare_3 :=, ValveFeedbackInputSelection :=, ValveFeedbackInput :=, Interlock := #Interlock, FBCheckDelay :=, WSCheckDelay :=, secs := "Sec_Pulse", AlarmAck :=, ModeSel :=, Fault :=, Reset :=, spare :=, spare_1 :=, spare_2 :=, OpFbTrip :=, OpWaterSensorTrip :=, FBCheckActualTime :=, WSCheckActualTime :=, Output =>, FeedBackTripAlarm =>, NoWaterFlowAlarm =>, LineColour =>, ValveColour =>, Mode =>, Status =>)
   END_RUNG
   // the same network as SCL:
   #Do05(AlwaysTrue := "AlwaysTRUE", AlwaysFalse := "AlwaysFALSE", Interlock := #Interlock, secs := "Sec_Pulse");   // "DigitalOutput"
END_REGION

